LIN {X -0.214,Y -606.391,Z 470.276,A 0.000,B 0.000,C 90.000,E1 265.698} C_DIS
LIN {X -0.037,Y -603.397,Z 470.269,A 0.000,B 0.000,C 90.000,E1 264.375} C_DIS
LIN {X 0.001,Y -599.105,Z 470.259,A 0.000,B 0.000,C 90.000,E1 262.534} C_DIS
LIN {X 0.083,Y -594.642,Z 470.248,A 0.000,B 0.000,C 90.000,E1 260.679} C_DIS
LIN {X 0.202,Y -591.268,Z 470.241,A 0.000,B 0.000,C 90.000,E1 259.342} C_DIS
LIN {X -0.200,Y -587.770,Z 470.234,A 0.000,B 0.000,C 90.000,E1 258.049} C_DIS
LIN {X 0.160,Y -583.456,Z 470.225,A 0.000,B 0.000,C 90.000,E1 256.408} C_DIS
LIN {X -0.227,Y -579.823,Z 470.217,A 0.000,B 0.000,C 90.000,E1 255.102} C_DIS
LIN {X -0.114,Y -576.110,Z 470.210,A 0.000,B 0.000,C 90.000,E1 253.740} C_DIS
LIN {X -0.279,Y -571.459,Z 470.201,A 0.000,B 0.000,C 90.000,E1 252.127} C_DIS
LIN {X 0.013,Y -567.401,Z 470.193,A 0.000,B 0.000,C 90.000,E1 250.732} C_DIS
LIN {X -0.299,Y -563.218,Z 470.185,A 0.000,B 0.000,C 90.000,E1 249.390} C_DIS
LIN {X 0.041,Y -558.827,Z 470.178,A 0.000,B 0.000,C 90.000,E1 247.975} C_DIS
LIN {X 0.000,Y -555.124,Z 470.172,A 0.000,B 0.000,C 90.000,E1 246.869} C_DIS
LIN {X -0.109,Y -550.348,Z 470.164,A 0.000,B 0.000,C 90.000,E1 245.485} C_DIS
LIN {X 0.182,Y -544.388,Z 470.154,A 0.000,B 0.000,C 90.000,E1 243.768} C_DIS
LIN {X 0.121,Y -539.419,Z 470.147,A 0.000,B 0.000,C 90.000,E1 242.359} C_DIS
LIN {X -0.063,Y -533.493,Z 470.137,A 0.000,B 0.000,C 90.000,E1 240.667} C_DIS
LIN {X -0.149,Y -526.505,Z 470.126,A 0.000,B 0.000,C 90.000,E1 238.663} C_DIS
LIN {X -0.079,Y -520.654,Z 470.116,A 0.000,B 0.000,C 90.000,E1 236.914} C_DIS
LIN {X -0.224,Y -515.720,Z 470.108,A 0.000,B 0.000,C 90.000,E1 235.468} C_DIS
LIN {X -0.088,Y -511.559,Z 470.102,A 0.000,B 0.000,C 90.000,E1 234.276} C_DIS
LIN {X -0.248,Y -499.683,Z 470.082,A 0.000,B 0.000,C 90.000,E1 230.723} C_DIS
LIN {X 0.150,Y -493.420,Z 470.070,A 0.000,B 0.000,C 90.000,E1 228.566} C_DIS
LIN {X 0.119,Y -486.466,Z 470.056,A 0.000,B 0.000,C 90.000,E1 226.134} C_DIS
LIN {X 0.299,Y -481.414,Z 470.046,A 0.000,B 0.000,C 90.000,E1 224.271} C_DIS
LIN {X 0.135,Y -475.759,Z 470.034,A 0.000,B 0.000,C 90.000,E1 222.123} C_DIS
LIN {X -0.016,Y -469.737,Z 470.020,A 0.000,B 0.000,C 90.000,E1 219.644} C_DIS
LIN {X -0.034,Y -464.806,Z 470.008,A 0.000,B 0.000,C 90.000,E1 217.443} C_DIS
LIN {X 0.021,Y -459.483,Z 469.994,A 0.000,B 0.000,C 90.000,E1 214.898} C_DIS
LIN {X -0.076,Y -455.045,Z 469.982,A 0.000,B 0.000,C 90.000,E1 212.673} C_DIS
LIN {X 0.035,Y -452.006,Z 469.973,A 0.000,B 0.000,C 90.000,E1 211.052} C_DIS
LIN {X -0.209,Y -447.757,Z 469.960,A 0.000,B 0.000,C 90.000,E1 208.821} C_DIS
LIN {X -0.083,Y -444.730,Z 469.951,A 0.000,B 0.000,C 90.000,E1 207.180} C_DIS
LIN {X 0.123,Y -442.265,Z 469.944,A 0.000,B 0.000,C 90.000,E1 205.848} C_DIS
LIN {X -0.108,Y -439.798,Z 469.936,A 0.000,B 0.000,C 90.000,E1 204.567} C_DIS
LIN {X -0.086,Y -435.424,Z 469.924,A 0.000,B 0.000,C 90.000,E1 202.259} C_DIS
LIN {X -0.097,Y -431.263,Z 469.911,A 0.000,B 0.000,C 90.000,E1 199.939} C_DIS
LIN {X 0.051,Y -427.360,Z 469.898,A 0.000,B 0.000,C 90.000,E1 197.583} C_DIS
LIN {X 0.032,Y -423.295,Z 469.883,A 0.000,B 0.000,C 90.000,E1 194.898} C_DIS
LIN {X 0.017,Y -420.092,Z 469.870,A 0.000,B 0.000,C 90.000,E1 192.535} C_DIS
LIN {X -0.153,Y -416.381,Z 469.853,A 0.000,B 0.000,C 90.000,E1 189.500} C_DIS
LIN {X 0.142,Y -413.690,Z 469.839,A 0.000,B 0.000,C 90.000,E1 187.068} C_DIS
LIN {X -0.160,Y -412.241,Z 469.832,A 0.000,B 0.000,C 90.000,E1 185.739} C_DIS
LIN {X -0.118,Y -410.914,Z 469.824,A 0.000,B 0.000,C 90.000,E1 184.359} C_DIS
LIN {X -0.131,Y -408.830,Z 469.811,A 0.000,B 0.000,C 90.000,E1 181.949} C_DIS
LIN {X 0.156,Y -406.733,Z 469.793,A 0.000,B 0.000,C 90.000,E1 178.797} C_DIS
LIN {X -0.003,Y -405.511,Z 469.778,A 0.000,B 0.000,C 90.000,E1 176.045} C_DIS
LIN {X -0.104,Y -404.848,Z 469.763,A 0.000,B 0.000,C 90.000,E1 173.280} C_DIS
LIN {X -0.104,Y -404.977,Z 469.745,A 0.000,B 0.000,C 90.000,E1 170.151} C_DIS
LIN {X 0.123,Y -405.882,Z 469.728,A 0.000,B 0.000,C 90.000,E1 166.992} C_DIS
LIN {X 0.056,Y -407.044,Z 469.714,A 0.000,B 0.000,C 90.000,E1 164.574} C_DIS
LIN {X -0.061,Y -409.699,Z 469.693,A 0.000,B 0.000,C 90.000,E1 160.786} C_DIS
LIN {X 0.053,Y -411.869,Z 469.680,A 0.000,B 0.000,C 90.000,E1 158.358} C_DIS
LIN {X -0.079,Y -414.415,Z 469.667,A 0.000,B 0.000,C 90.000,E1 155.973} C_DIS
LIN {X -0.204,Y -416.381,Z 469.657,A 0.000,B 0.000,C 90.000,E1 154.280} C_DIS
LIN {X 0.107,Y -419.671,Z 469.642,A 0.000,B 0.000,C 90.000,E1 151.513} C_DIS
LIN {X 0.075,Y -421.752,Z 469.632,A 0.000,B 0.000,C 90.000,E1 149.822} C_DIS
LIN {X 0.146,Y -423.876,Z 469.623,A 0.000,B 0.000,C 90.000,E1 148.122} C_DIS
LIN {X -0.101,Y -426.458,Z 469.612,A 0.000,B 0.000,C 90.000,E1 146.135} C_DIS
LIN {X -0.048,Y -429.095,Z 469.601,A 0.000,B 0.000,C 90.000,E1 144.116} C_DIS
LIN {X 0.071,Y -430.982,Z 469.593,A 0.000,B 0.000,C 90.000,E1 142.763} C_DIS
LIN {X -0.214,Y -433.774,Z 469.582,A 0.000,B 0.000,C 90.000,E1 140.803} C_DIS
LIN {X -0.095,Y -435.681,Z 469.575,A 0.000,B 0.000,C 90.000,E1 139.461} C_DIS
LIN {X -0.003,Y -437.965,Z 469.566,A 0.000,B 0.000,C 90.000,E1 137.796} C_DIS
LIN {X 0.104,Y -440.095,Z 469.556,A 0.000,B 0.000,C 90.000,E1 136.134} C_DIS
LIN {X 0.001,Y -441.095,Z 469.551,A 0.000,B 0.000,C 90.000,E1 135.162} C_DIS
LIN {X -0.119,Y -442.209,Z 469.544,A 0.000,B 0.000,C 90.000,E1 133.866} C_DIS
LIN {X 0.095,Y -442.966,Z 469.536,A 0.000,B 0.000,C 90.000,E1 132.528} C_DIS
LIN {X 0.022,Y -443.267,Z 469.529,A 0.000,B 0.000,C 90.000,E1 131.229} C_DIS
LIN {X -0.017,Y -443.139,Z 469.524,A 0.000,B 0.000,C 90.000,E1 130.253} C_DIS
LIN {X -0.058,Y -442.518,Z 469.518,A 0.000,B 0.000,C 90.000,E1 129.277} C_DIS
LIN {X -0.110,Y -441.689,Z 469.513,A 0.000,B 0.000,C 90.000,E1 128.302} C_DIS
LIN {X -0.097,Y -440.525,Z 469.507,A 0.000,B 0.000,C 90.000,E1 127.317} C_DIS
LIN {X -0.155,Y -438.561,Z 469.500,A 0.000,B 0.000,C 90.000,E1 126.011} C_DIS
LIN {X 0.158,Y -437.427,Z 469.496,A 0.000,B 0.000,C 90.000,E1 125.311} C_DIS
LIN {X 0.148,Y -434.935,Z 469.489,A 0.000,B 0.000,C 90.000,E1 123.992} C_DIS
LIN {X 0.094,Y -432.035,Z 469.482,A 0.000,B 0.000,C 90.000,E1 122.673} C_DIS
LIN {X -0.005,Y -428.435,Z 469.473,A 0.000,B 0.000,C 90.000,E1 121.052} C_DIS
LIN {X -0.045,Y -428.429,Z 469.473,A 0.000,B 0.000,C 90.000,E1 121.052} C_DIS
LIN {X 0.121,Y -430.573,Z 469.469,A 0.000,B 0.000,C 90.000,E1 120.335} C_DIS
LIN {X -0.079,Y -441.483,Z 469.445,A 0.000,B 0.000,C 90.000,E1 116.052} C_DIS
LIN {X -0.159,Y -444.396,Z 469.439,A 0.000,B 0.000,C 90.000,E1 115.079} C_DIS
LIN {X 0.098,Y -445.208,Z 469.437,A 0.000,B 0.000,C 90.000,E1 114.719} C_DIS
LIN {X -0.040,Y -454.406,Z 469.416,A 0.000,B 0.000,C 90.000,E1 110.844} C_DIS
LIN {X -0.081,Y -457.079,Z 469.410,A 0.000,B 0.000,C 90.000,E1 109.885} C_DIS
LIN {X 0.004,Y -461.437,Z 469.398,A 0.000,B 0.000,C 90.000,E1 107.638} C_DIS
LIN {X -0.276,Y -467.270,Z 469.384,A 0.000,B 0.000,C 90.000,E1 105.134} C_DIS
LIN {X 0.101,Y -467.963,Z 469.382,A 0.000,B 0.000,C 90.000,E1 104.773} C_DIS
LIN {X -0.171,Y -476.219,Z 469.356,A 0.000,B 0.000,C 90.000,E1 100.074} C_DIS
LIN {X -0.091,Y -476.372,Z 469.355,A 0.000,B 0.000,C 90.000,E1 99.905} C_DIS
LIN {X -0.148,Y -526.605,Z 469.355,A 0.000,B 0.000,C 90.000,E1 99.905} C_DIS
LIN {X -0.102,Y -537.151,Z 469.355,A 0.000,B 0.000,C 90.000,E1 99.849} C_DIS
LIN {X 0.113,Y -540.500,Z 469.355,A 0.000,B 0.000,C 90.000,E1 99.792} C_DIS
LIN {X -0.208,Y -553.262,Z 469.353,A 0.000,B 0.000,C 90.000,E1 99.613} C_DIS
LIN {X 0.013,Y -559.633,Z 469.353,A 0.000,B 0.000,C 90.000,E1 99.443} C_DIS
LIN {X 0.063,Y -566.108,Z 469.352,A 0.000,B 0.000,C 90.000,E1 99.265} C_DIS
LIN {X 0.294,Y -576.120,Z 469.350,A 0.000,B 0.000,C 90.000,E1 98.916} C_DIS
LIN {X 0.150,Y -582.565,Z 469.348,A 0.000,B 0.000,C 90.000,E1 98.690} C_DIS
LIN {X 0.006,Y -592.233,Z 469.346,A 0.000,B 0.000,C 90.000,E1 98.276} C_DIS
LIN {X -0.304,Y -598.318,Z 469.344,A 0.000,B 0.000,C 90.000,E1 97.992} C_DIS
LIN {X -0.023,Y -601.041,Z 469.343,A 0.000,B 0.000,C 90.000,E1 97.814} C_DIS
LIN {X 0.102,Y -605.450,Z 469.342,A 0.000,B 0.000,C 90.000,E1 97.530} C_DIS
LIN {X 0.141,Y -611.163,Z 469.340,A 0.000,B 0.000,C 90.000,E1 97.125} C_DIS
LIN {X -0.132,Y -616.701,Z 469.337,A 0.000,B 0.000,C 90.000,E1 96.720} C_DIS
LIN {X -0.210,Y -623.076,Z 469.334,A 0.000,B 0.000,C 90.000,E1 96.144} C_DIS
LIN {X 0.323,Y -625.293,Z 469.333,A 0.000,B 0.000,C 90.000,E1 95.853} C_DIS
LIN {X -0.209,Y -629.691,Z 469.330,A 0.000,B 0.000,C 90.000,E1 95.391} C_DIS
LIN {X 0.002,Y -636.399,Z 469.324,A 0.000,B 0.000,C 90.000,E1 94.359} C_DIS
LIN {X 0.296,Y -638.500,Z 469.322,A 0.000,B 0.000,C 90.000,E1 93.955} C_DIS
LIN {X -0.083,Y -640.476,Z 469.320,A 0.000,B 0.000,C 90.000,E1 93.612} C_DIS
LIN {X 0.106,Y -642.677,Z 469.317,A 0.000,B 0.000,C 90.000,E1 93.094} C_DIS
LIN {X -0.135,Y -643.601,Z 469.316,A 0.000,B 0.000,C 90.000,E1 92.865} C_DIS
LIN {X 0.040,Y -645.162,Z 469.313,A 0.000,B 0.000,C 90.000,E1 92.350} C_DIS
LIN {X 0.232,Y -646.453,Z 469.310,A 0.000,B 0.000,C 90.000,E1 91.835} C_DIS
LIN {X -0.196,Y -647.322,Z 469.308,A 0.000,B 0.000,C 90.000,E1 91.375} C_DIS
LIN {X 0.010,Y -647.929,Z 469.305,A 0.000,B 0.000,C 90.000,E1 90.859} C_DIS
LIN {X -0.207,Y -648.173,Z 469.303,A 0.000,B 0.000,C 90.000,E1 90.630} C_DIS
LIN {X 0.008,Y -648.223,Z 469.301,A 0.000,B 0.000,C 90.000,E1 90.115} C_DIS
LIN {X 0.224,Y -647.934,Z 469.298,A 0.000,B 0.000,C 90.000,E1 89.599} C_DIS
LIN {X -0.209,Y -647.327,Z 469.295,A 0.000,B 0.000,C 90.000,E1 89.141} C_DIS
LIN {X 0.219,Y -646.938,Z 469.294,A 0.000,B 0.000,C 90.000,E1 88.854} C_DIS
LIN {X -0.221,Y -645.753,Z 469.291,A 0.000,B 0.000,C 90.000,E1 88.396} C_DIS
LIN {X -0.002,Y -644.242,Z 469.288,A 0.000,B 0.000,C 90.000,E1 87.879} C_DIS
LIN {X -0.228,Y -643.391,Z 469.287,A 0.000,B 0.000,C 90.000,E1 87.650} C_DIS
LIN {X -0.048,Y -641.396,Z 469.284,A 0.000,B 0.000,C 90.000,E1 87.135} C_DIS
LIN {X 0.151,Y -638.859,Z 469.281,A 0.000,B 0.000,C 90.000,E1 86.617} C_DIS
LIN {X 0.079,Y -634.722,Z 469.277,A 0.000,B 0.000,C 90.000,E1 85.869} C_DIS
LIN {X -0.173,Y -628.526,Z 469.272,A 0.000,B 0.000,C 90.000,E1 85.008} C_DIS
LIN {X -0.201,Y -623.501,Z 469.269,A 0.000,B 0.000,C 90.000,E1 84.375} C_DIS
LIN {X 0.184,Y -616.636,Z 469.264,A 0.000,B 0.000,C 90.000,E1 83.571} C_DIS
LIN {X -0.211,Y -611.344,Z 469.262,A 0.000,B 0.000,C 90.000,E1 83.109} C_DIS
LIN {X 0.221,Y -605.741,Z 469.259,A 0.000,B 0.000,C 90.000,E1 82.591} C_DIS
LIN {X -0.255,Y -599.923,Z 469.257,A 0.000,B 0.000,C 90.000,E1 82.186} C_DIS
LIN {X -0.109,Y -596.254,Z 469.255,A 0.000,B 0.000,C 90.000,E1 81.951} C_DIS
LIN {X -0.224,Y -593.898,Z 469.254,A 0.000,B 0.000,C 90.000,E1 81.781} C_DIS
LIN {X 0.017,Y -588.144,Z 469.252,A 0.000,B 0.000,C 90.000,E1 81.376} C_DIS
LIN {X -0.178,Y -584.150,Z 469.251,A 0.000,B 0.000,C 90.000,E1 81.197} C_DIS
LIN {X -0.046,Y -581.425,Z 469.250,A 0.000,B 0.000,C 90.000,E1 81.027} C_DIS
LIN {X -0.280,Y -575.599,Z 469.249,A 0.000,B 0.000,C 90.000,E1 80.792} C_DIS
LIN {X 0.043,Y -570.052,Z 469.248,A 0.000,B 0.000,C 90.000,E1 80.557} C_DIS
LIN {X 0.000,Y -563.805,Z 469.247,A 0.000,B 0.000,C 90.000,E1 80.387} C_DIS
LIN {X -0.304,Y -559.346,Z 469.246,A 0.000,B 0.000,C 90.000,E1 80.330} C_DIS
LIN {X -0.278,Y -556.297,Z 469.246,A 0.000,B 0.000,C 90.000,E1 80.274} C_DIS
LIN {X -0.067,Y -550.275,Z 469.246,A 0.000,B 0.000,C 90.000,E1 80.208} C_DIS
LIN {X -0.089,Y -483.137,Z 469.246,A 0.000,B 0.000,C 90.000,E1 80.208} C_DIS
LIN {X -0.081,Y -480.607,Z 469.228,A 0.000,B 0.000,C 90.000,E1 76.992} C_DIS
LIN {X -0.223,Y -480.245,Z 469.226,A 0.000,B 0.000,C 90.000,E1 76.700} C_DIS
LIN {X 0.134,Y -474.075,Z 469.200,A 0.000,B 0.000,C 90.000,E1 72.000} C_DIS
LIN {X 0.163,Y -465.515,Z 469.172,A 0.000,B 0.000,C 90.000,E1 66.975} C_DIS
LIN {X 0.094,Y -456.793,Z 469.148,A 0.000,B 0.000,C 90.000,E1 62.692} C_DIS
LIN {X 0.032,Y -456.650,Z 469.148,A 0.000,B 0.000,C 90.000,E1 62.615} C_DIS
LIN {X -0.008,Y -456.674,Z 469.148,A 0.000,B 0.000,C 90.000,E1 62.615} C_DIS
LIN {X 0.088,Y -465.116,Z 469.140,A 0.000,B 0.000,C 90.000,E1 61.257} C_DIS
LIN {X 0.137,Y -469.919,Z 469.136,A 0.000,B 0.000,C 90.000,E1 60.461} C_DIS
LIN {X 0.232,Y -474.530,Z 469.132,A 0.000,B 0.000,C 90.000,E1 59.665} C_DIS
LIN {X -0.035,Y -478.623,Z 469.127,A 0.000,B 0.000,C 90.000,E1 58.918} C_DIS
LIN {X -0.065,Y -480.940,Z 469.125,A 0.000,B 0.000,C 90.000,E1 58.456} C_DIS
LIN {X -0.050,Y -483.692,Z 469.121,A 0.000,B 0.000,C 90.000,E1 57.837} C_DIS
LIN {X -0.276,Y -486.044,Z 469.118,A 0.000,B 0.000,C 90.000,E1 57.248} C_DIS
LIN {X 0.007,Y -489.125,Z 469.113,A 0.000,B 0.000,C 90.000,E1 56.294} C_DIS
LIN {X -0.080,Y -491.318,Z 469.108,A 0.000,B 0.000,C 90.000,E1 55.388} C_DIS
LIN {X 0.010,Y -492.589,Z 469.104,A 0.000,B 0.000,C 90.000,E1 54.769} C_DIS
LIN {X -0.040,Y -494.001,Z 469.099,A 0.000,B 0.000,C 90.000,E1 53.863} C_DIS
LIN {X 0.216,Y -494.947,Z 469.094,A 0.000,B 0.000,C 90.000,E1 52.924} C_DIS
LIN {X 0.096,Y -495.629,Z 469.089,A 0.000,B 0.000,C 90.000,E1 52.029} C_DIS
LIN {X 0.066,Y -496.085,Z 469.084,A 0.000,B 0.000,C 90.000,E1 51.126} C_DIS
LIN {X -0.041,Y -496.341,Z 469.079,A 0.000,B 0.000,C 90.000,E1 50.231} C_DIS
LIN {X 0.179,Y -496.434,Z 469.074,A 0.000,B 0.000,C 90.000,E1 49.299} C_DIS
LIN {X 0.264,Y -496.318,Z 469.067,A 0.000,B 0.000,C 90.000,E1 48.081} C_DIS
LIN {X -0.209,Y -496.105,Z 469.062,A 0.000,B 0.000,C 90.000,E1 47.229} C_DIS
LIN {X 0.202,Y -495.692,Z 469.056,A 0.000,B 0.000,C 90.000,E1 45.972} C_DIS
LIN {X -0.263,Y -495.039,Z 469.047,A 0.000,B 0.000,C 90.000,E1 44.514} C_DIS
LIN {X -0.047,Y -494.218,Z 469.039,A 0.000,B 0.000,C 90.000,E1 42.975} C_DIS
LIN {X -0.157,Y -493.082,Z 469.030,A 0.000,B 0.000,C 90.000,E1 41.472} C_DIS
LIN {X 0.042,Y -491.981,Z 469.022,A 0.000,B 0.000,C 90.000,E1 39.930} C_DIS
LIN {X 0.118,Y -490.517,Z 469.012,A 0.000,B 0.000,C 90.000,E1 38.096} C_DIS
LIN {X 0.180,Y -489.507,Z 469.005,A 0.000,B 0.000,C 90.000,E1 36.870} C_DIS
LIN {X -0.064,Y -488.412,Z 468.998,A 0.000,B 0.000,C 90.000,E1 35.678} C_DIS
LIN {X -0.044,Y -487.237,Z 468.991,A 0.000,B 0.000,C 90.000,E1 34.452} C_DIS
LIN {X 0.042,Y -485.625,Z 468.983,A 0.000,B 0.000,C 90.000,E1 32.911} C_DIS
LIN {X 0.178,Y -483.531,Z 468.973,A 0.000,B 0.000,C 90.000,E1 31.052} C_DIS
LIN {X -0.261,Y -482.018,Z 468.966,A 0.000,B 0.000,C 90.000,E1 29.873} C_DIS
LIN {X 0.123,Y -479.814,Z 468.956,A 0.000,B 0.000,C 90.000,E1 27.975} C_DIS
LIN {X -0.223,Y -477.343,Z 468.944,A 0.000,B 0.000,C 90.000,E1 25.848} C_DIS
LIN {X -0.057,Y -474.460,Z 468.926,A 0.000,B 0.000,C 90.000,E1 22.717} C_DIS
LIN {X 0.121,Y -472.524,Z 468.911,A 0.000,B 0.000,C 90.000,E1 19.885} C_DIS
LIN {X 0.136,Y -471.211,Z 468.898,A 0.000,B 0.000,C 90.000,E1 17.692} C_DIS
LIN {X -0.128,Y -470.067,Z 468.888,A 0.000,B 0.000,C 90.000,E1 15.843} C_DIS
LIN {X 0.120,Y -468.728,Z 468.874,A 0.000,B 0.000,C 90.000,E1 13.300} C_DIS
LIN {X -0.251,Y -467.699,Z 468.857,A 0.000,B 0.000,C 90.000,E1 10.197} C_DIS
LIN {X 0.012,Y -467.337,Z 468.843,A 0.000,B 0.000,C 90.000,E1 7.644} C_DIS
LIN {X -0.078,Y -467.737,Z 468.823,A 0.000,B 0.000,C 90.000,E1 4.188} C_DIS
LIN {X 0.227,Y -469.374,Z 468.804,A 0.000,B 0.000,C 90.000,E1 0.688} C_DIS
LIN {X -0.218,Y -471.580,Z 468.788,A 0.000,B 0.000,C 90.000,E1 357.936} C_DIS
LIN {X -0.048,Y -474.192,Z 468.775,A 0.000,B 0.000,C 90.000,E1 355.412} C_DIS
LIN {X -0.151,Y -477.274,Z 468.761,A 0.000,B 0.000,C 90.000,E1 352.932} C_DIS
LIN {X 0.095,Y -481.700,Z 468.743,A 0.000,B 0.000,C 90.000,E1 349.803} C_DIS
LIN {X -0.184,Y -490.068,Z 468.718,A 0.000,B 0.000,C 90.000,E1 345.227} C_DIS
LIN {X -0.060,Y -495.409,Z 468.704,A 0.000,B 0.000,C 90.000,E1 342.779} C_DIS
LIN {X -0.063,Y -499.708,Z 468.694,A 0.000,B 0.000,C 90.000,E1 340.967} C_DIS
LIN {X 0.121,Y -503.389,Z 468.686,A 0.000,B 0.000,C 90.000,E1 339.444} C_DIS
LIN {X -0.103,Y -507.108,Z 468.678,A 0.000,B 0.000,C 90.000,E1 337.975} C_DIS
LIN {X -0.073,Y -510.736,Z 468.669,A 0.000,B 0.000,C 90.000,E1 336.485} C_DIS
LIN {X -0.213,Y -512.934,Z 468.664,A 0.000,B 0.000,C 90.000,E1 335.613} C_DIS
LIN {X 0.125,Y -516.463,Z 468.656,A 0.000,B 0.000,C 90.000,E1 334.101} C_DIS
LIN {X -0.166,Y -520.033,Z 468.648,A 0.000,B 0.000,C 90.000,E1 332.666} C_DIS
LIN {X 0.078,Y -523.580,Z 468.640,A 0.000,B 0.000,C 90.000,E1 331.179} C_DIS
LIN {X -0.126,Y -527.898,Z 468.630,A 0.000,B 0.000,C 90.000,E1 329.459} C_DIS
LIN {X 0.039,Y -532.324,Z 468.621,A 0.000,B 0.000,C 90.000,E1 327.709} C_DIS
LIN {X -0.153,Y -537.489,Z 468.610,A 0.000,B 0.000,C 90.000,E1 325.722} C_DIS
LIN {X 0.040,Y -541.224,Z 468.602,A 0.000,B 0.000,C 90.000,E1 324.276} C_DIS
LIN {X 0.208,Y -545.829,Z 468.592,A 0.000,B 0.000,C 90.000,E1 322.557} C_DIS
LIN {X 0.044,Y -550.377,Z 468.583,A 0.000,B 0.000,C 90.000,E1 320.884} C_DIS
LIN {X -0.101,Y -554.896,Z 468.573,A 0.000,B 0.000,C 90.000,E1 319.218} C_DIS
LIN {X 0.303,Y -560.197,Z 468.563,A 0.000,B 0.000,C 90.000,E1 317.229} C_DIS
LIN {X 0.013,Y -565.320,Z 468.552,A 0.000,B 0.000,C 90.000,E1 315.324} C_DIS
LIN {X -0.259,Y -569.637,Z 468.543,A 0.000,B 0.000,C 90.000,E1 313.704} C_DIS
LIN {X -0.248,Y -572.591,Z 468.537,A 0.000,B 0.000,C 90.000,E1 312.609} C_DIS
LIN {X 0.084,Y -576.826,Z 468.528,A 0.000,B 0.000,C 90.000,E1 310.943} C_DIS
LIN {X 0.064,Y -581.088,Z 468.519,A 0.000,B 0.000,C 90.000,E1 309.322} C_DIS
LIN {X -0.166,Y -585.312,Z 468.510,A 0.000,B 0.000,C 90.000,E1 307.729} C_DIS
LIN {X -0.033,Y -588.807,Z 468.502,A 0.000,B 0.000,C 90.000,E1 306.377} C_DIS
LIN {X 0.035,Y -592.869,Z 468.493,A 0.000,B 0.000,C 90.000,E1 304.771} C_DIS
LIN {X -0.036,Y -596.152,Z 468.486,A 0.000,B 0.000,C 90.000,E1 303.452} C_DIS
LIN {X -0.288,Y -598.661,Z 468.480,A 0.000,B 0.000,C 90.000,E1 302.418} C_DIS
LIN {X -0.004,Y -601.106,Z 468.474,A 0.000,B 0.000,C 90.000,E1 301.337} C_DIS
LIN {X 0.242,Y -603.935,Z 468.467,A 0.000,B 0.000,C 90.000,E1 300.001} C_DIS
LIN {X 0.293,Y -606.023,Z 468.461,A 0.000,B 0.000,C 90.000,E1 298.949} C_DIS
LIN {X 0.369,Y -607.930,Z 468.455,A 0.000,B 0.000,C 90.000,E1 297.897} C_DIS
LIN {X 0.066,Y -611.293,Z 468.445,A 0.000,B 0.000,C 90.000,E1 296.104} C_DIS
LIN {X -0.040,Y -612.586,Z 468.441,A 0.000,B 0.000,C 90.000,E1 295.335} C_DIS
LIN {X 0.107,Y -614.428,Z 468.434,A 0.000,B 0.000,C 90.000,E1 294.027} C_DIS
LIN {X 0.244,Y -616.844,Z 468.424,A 0.000,B 0.000,C 90.000,E1 292.206} C_DIS
LIN {X 0.236,Y -618.384,Z 468.416,A 0.000,B 0.000,C 90.000,E1 290.918} C_DIS
LIN {X 0.017,Y -620.101,Z 468.408,A 0.000,B 0.000,C 90.000,E1 289.396} C_DIS
LIN {X -0.174,Y -621.635,Z 468.399,A 0.000,B 0.000,C 90.000,E1 287.873} C_DIS
LIN {X 0.058,Y -623.055,Z 468.391,A 0.000,B 0.000,C 90.000,E1 286.315} C_DIS
LIN {X -0.245,Y -624.059,Z 468.384,A 0.000,B 0.000,C 90.000,E1 285.064} C_DIS
LIN {X 0.124,Y -624.729,Z 468.378,A 0.000,B 0.000,C 90.000,E1 284.008} C_DIS
LIN {X 0.101,Y -625.512,Z 468.369,A 0.000,B 0.000,C 90.000,E1 282.479} C_DIS
LIN {X 0.293,Y -625.911,Z 468.362,A 0.000,B 0.000,C 90.000,E1 281.186} C_DIS
LIN {X -0.252,Y -626.151,Z 468.355,A 0.000,B 0.000,C 90.000,E1 279.962} C_DIS
LIN {X 0.128,Y -625.966,Z 468.347,A 0.000,B 0.000,C 90.000,E1 278.398} C_DIS
LIN {X -0.215,Y -625.694,Z 468.341,A 0.000,B 0.000,C 90.000,E1 277.409} C_DIS
LIN {X 0.202,Y -625.319,Z 468.337,A 0.000,B 0.000,C 90.000,E1 276.606} C_DIS
LIN {X -0.231,Y -624.667,Z 468.331,A 0.000,B 0.000,C 90.000,E1 275.625} C_DIS
LIN {X 0.270,Y -623.439,Z 468.324,A 0.000,B 0.000,C 90.000,E1 274.302} C_DIS
LIN {X -0.241,Y -622.206,Z 468.318,A 0.000,B 0.000,C 90.000,E1 273.326} C_DIS
LIN {X -0.147,Y -620.769,Z 468.313,A 0.000,B 0.000,C 90.000,E1 272.293} C_DIS
LIN {X -0.079,Y -619.105,Z 468.307,A 0.000,B 0.000,C 90.000,E1 271.260} C_DIS
LIN {X 0.262,Y -616.863,Z 468.300,A 0.000,B 0.000,C 90.000,E1 269.943} C_DIS
LIN {X 0.246,Y -613.920,Z 468.291,A 0.000,B 0.000,C 90.000,E1 268.396} C_DIS
LIN {X 0.219,Y -611.803,Z 468.286,A 0.000,B 0.000,C 90.000,E1 267.364} C_DIS
LIN {X 0.166,Y -609.594,Z 468.280,A 0.000,B 0.000,C 90.000,E1 266.331} C_DIS
LIN {X -0.186,Y -607.893,Z 468.275,A 0.000,B 0.000,C 90.000,E1 265.584} C_DIS
LIN {X 0.014,Y -604.843,Z 468.268,A 0.000,B 0.000,C 90.000,E1 264.261} C_DIS
LIN {X -0.143,Y -601.122,Z 468.259,A 0.000,B 0.000,C 90.000,E1 262.704} C_DIS
LIN {X 0.294,Y -597.231,Z 468.251,A 0.000,B 0.000,C 90.000,E1 261.084} C_DIS
LIN {X -0.125,Y -593.897,Z 468.243,A 0.000,B 0.000,C 90.000,E1 259.803} C_DIS
LIN {X 0.249,Y -589.648,Z 468.234,A 0.000,B 0.000,C 90.000,E1 258.173} C_DIS
LIN {X 0.069,Y -585.249,Z 468.226,A 0.000,B 0.000,C 90.000,E1 256.589} C_DIS
LIN {X -0.063,Y -580.830,Z 468.217,A 0.000,B 0.000,C 90.000,E1 254.991} C_DIS
LIN {X -0.150,Y -577.822,Z 468.211,A 0.000,B 0.000,C 90.000,E1 253.921} C_DIS
LIN {X -0.280,Y -573.149,Z 468.202,A 0.000,B 0.000,C 90.000,E1 252.308} C_DIS
LIN {X -0.150,Y -568.232,Z 468.193,A 0.000,B 0.000,C 90.000,E1 250.659} C_DIS
LIN {X 0.090,Y -563.988,Z 468.185,A 0.000,B 0.000,C 90.000,E1 249.263} C_DIS
LIN {X -0.075,Y -559.589,Z 468.177,A 0.000,B 0.000,C 90.000,E1 247.901} C_DIS
LIN {X -0.098,Y -555.824,Z 468.171,A 0.000,B 0.000,C 90.000,E1 246.794} C_DIS
LIN {X -0.187,Y -551.005,Z 468.163,A 0.000,B 0.000,C 90.000,E1 245.409} C_DIS
LIN {X -0.115,Y -545.003,Z 468.154,A 0.000,B 0.000,C 90.000,E1 243.717} C_DIS
LIN {X 0.092,Y -541.007,Z 468.148,A 0.000,B 0.000,C 90.000,E1 242.564} C_DIS
LIN {X 0.197,Y -535.050,Z 468.138,A 0.000,B 0.000,C 90.000,E1 240.845} C_DIS
LIN {X 0.185,Y -529.009,Z 468.129,A 0.000,B 0.000,C 90.000,E1 239.125} C_DIS
LIN {X -0.063,Y -521.138,Z 468.116,A 0.000,B 0.000,C 90.000,E1 236.834} C_DIS
LIN {X -0.196,Y -516.196,Z 468.108,A 0.000,B 0.000,C 90.000,E1 235.388} C_DIS
LIN {X -0.127,Y -510.971,Z 468.099,A 0.000,B 0.000,C 90.000,E1 233.909} C_DIS
LIN {X -0.306,Y -499.239,Z 468.080,A 0.000,B 0.000,C 90.000,E1 230.356} C_DIS
LIN {X -0.143,Y -493.865,Z 468.070,A 0.000,B 0.000,C 90.000,E1 228.528} C_DIS
LIN {X 0.210,Y -486.936,Z 468.056,A 0.000,B 0.000,C 90.000,E1 226.053} C_DIS
LIN {X -0.282,Y -481.901,Z 468.046,A 0.000,B 0.000,C 90.000,E1 224.271} C_DIS
LIN {X 0.035,Y -475.440,Z 468.032,A 0.000,B 0.000,C 90.000,E1 221.757} C_DIS
LIN {X 0.105,Y -470.205,Z 468.020,A 0.000,B 0.000,C 90.000,E1 219.564} C_DIS
LIN {X 0.097,Y -465.261,Z 468.008,A 0.000,B 0.000,C 90.000,E1 217.363} C_DIS
LIN {X 0.039,Y -460.593,Z 467.995,A 0.000,B 0.000,C 90.000,E1 215.152} C_DIS
LIN {X -0.287,Y -456.091,Z 467.983,A 0.000,B 0.000,C 90.000,E1 212.959} C_DIS
LIN {X -0.051,Y -452.410,Z 467.972,A 0.000,B 0.000,C 90.000,E1 211.003} C_DIS
LIN {X -0.136,Y -448.780,Z 467.961,A 0.000,B 0.000,C 90.000,E1 209.077} C_DIS
LIN {X -0.134,Y -445.153,Z 467.951,A 0.000,B 0.000,C 90.000,E1 207.129} C_DIS
LIN {X 0.128,Y -442.052,Z 467.942,A 0.000,B 0.000,C 90.000,E1 205.463} C_DIS
LIN {X 0.134,Y -438.893,Z 467.932,A 0.000,B 0.000,C 90.000,E1 203.823} C_DIS
LIN {X -0.029,Y -434.559,Z 467.920,A 0.000,B 0.000,C 90.000,E1 201.535} C_DIS
LIN {X 0.130,Y -430.992,Z 467.909,A 0.000,B 0.000,C 90.000,E1 199.523} C_DIS
LIN {X 0.198,Y -427.662,Z 467.897,A 0.000,B 0.000,C 90.000,E1 197.511} C_DIS
LIN {X 0.174,Y -423.572,Z 467.883,A 0.000,B 0.000,C 90.000,E1 194.828} C_DIS
LIN {X -0.009,Y -420.793,Z 467.871,A 0.000,B 0.000,C 90.000,E1 192.827} C_DIS
LIN {X -0.155,Y -417.027,Z 467.854,A 0.000,B 0.000,C 90.000,E1 189.792} C_DIS
LIN {X 0.216,Y -414.290,Z 467.841,A 0.000,B 0.000,C 90.000,E1 187.352} C_DIS
LIN {X -0.089,Y -412.479,Z 467.832,A 0.000,B 0.000,C 90.000,E1 185.682} C_DIS
LIN {X -0.029,Y -410.479,Z 467.820,A 0.000,B 0.000,C 90.000,E1 183.612} C_DIS
LIN {X -0.060,Y -408.513,Z 467.807,A 0.000,B 0.000,C 90.000,E1 181.203} C_DIS
LIN {X 0.196,Y -406.406,Z 467.787,A 0.000,B 0.000,C 90.000,E1 177.707} C_DIS
LIN {X 0.058,Y -405.485,Z 467.774,A 0.000,B 0.000,C 90.000,E1 175.298} C_DIS
LIN {X -0.029,Y -405.073,Z 467.753,A 0.000,B 0.000,C 90.000,E1 171.489} C_DIS
LIN {X 0.117,Y -405.657,Z 467.735,A 0.000,B 0.000,C 90.000,E1 168.342} C_DIS
LIN {X 0.060,Y -407.016,Z 467.718,A 0.000,B 0.000,C 90.000,E1 165.227} C_DIS
LIN {X -0.186,Y -409.477,Z 467.697,A 0.000,B 0.000,C 90.000,E1 161.456} C_DIS
LIN {X -0.076,Y -411.606,Z 467.683,A 0.000,B 0.000,C 90.000,E1 159.028} C_DIS
LIN {X -0.130,Y -413.707,Z 467.672,A 0.000,B 0.000,C 90.000,E1 156.975} C_DIS
LIN {X 0.178,Y -416.475,Z 467.659,A 0.000,B 0.000,C 90.000,E1 154.537} C_DIS
LIN {X -0.074,Y -419.770,Z 467.644,A 0.000,B 0.000,C 90.000,E1 151.847} C_DIS
LIN {X 0.104,Y -421.897,Z 467.634,A 0.000,B 0.000,C 90.000,E1 150.127} C_DIS
LIN {X -0.079,Y -424.935,Z 467.621,A 0.000,B 0.000,C 90.000,E1 147.788} C_DIS
LIN {X 0.049,Y -427.605,Z 467.610,A 0.000,B 0.000,C 90.000,E1 145.754} C_DIS
LIN {X 0.014,Y -430.884,Z 467.597,A 0.000,B 0.000,C 90.000,E1 143.417} C_DIS
LIN {X -0.010,Y -434.217,Z 467.584,A 0.000,B 0.000,C 90.000,E1 141.090} C_DIS
LIN {X -0.223,Y -436.669,Z 467.575,A 0.000,B 0.000,C 90.000,E1 139.461} C_DIS
LIN {X -0.111,Y -439.101,Z 467.565,A 0.000,B 0.000,C 90.000,E1 137.796} C_DIS
LIN {X 0.018,Y -441.323,Z 467.556,A 0.000,B 0.000,C 90.000,E1 136.134} C_DIS
LIN {X -0.097,Y -442.713,Z 467.549,A 0.000,B 0.000,C 90.000,E1 134.838} C_DIS
LIN {X -0.147,Y -443.338,Z 467.545,A 0.000,B 0.000,C 90.000,E1 134.190} C_DIS
LIN {X 0.108,Y -444.040,Z 467.540,A 0.000,B 0.000,C 90.000,E1 133.176} C_DIS
LIN {X 0.045,Y -444.514,Z 467.535,A 0.000,B 0.000,C 90.000,E1 132.204} C_DIS
LIN {X 0.015,Y -444.787,Z 467.529,A 0.000,B 0.000,C 90.000,E1 131.229} C_DIS
LIN {X -0.007,Y -444.703,Z 467.524,A 0.000,B 0.000,C 90.000,E1 130.253} C_DIS
LIN {X -0.060,Y -443.919,Z 467.516,A 0.000,B 0.000,C 90.000,E1 128.955} C_DIS
LIN {X -0.025,Y -443.006,Z 467.511,A 0.000,B 0.000,C 90.000,E1 127.971} C_DIS
LIN {X -0.077,Y -441.762,Z 467.506,A 0.000,B 0.000,C 90.000,E1 126.996} C_DIS
LIN {X -0.060,Y -440.315,Z 467.500,A 0.000,B 0.000,C 90.000,E1 126.011} C_DIS
LIN {X -0.090,Y -439.161,Z 467.496,A 0.000,B 0.000,C 90.000,E1 125.358} C_DIS
LIN {X -0.079,Y -436.596,Z 467.489,A 0.000,B 0.000,C 90.000,E1 124.040} C_DIS
LIN {X -0.002,Y -434.413,Z 467.484,A 0.000,B 0.000,C 90.000,E1 123.038} C_DIS
LIN {X -0.057,Y -430.655,Z 467.474,A 0.000,B 0.000,C 90.000,E1 121.386} C_DIS
LIN {X -0.127,Y -429.254,Z 467.471,A 0.000,B 0.000,C 90.000,E1 120.797} C_DIS
LIN {X -0.166,Y -429.257,Z 467.471,A 0.000,B 0.000,C 90.000,E1 120.797} C_DIS
LIN {X -0.048,Y -430.488,Z 467.469,A 0.000,B 0.000,C 90.000,E1 120.384} C_DIS
LIN {X -0.255,Y -432.832,Z 467.463,A 0.000,B 0.000,C 90.000,E1 119.411} C_DIS
LIN {X 0.160,Y -442.358,Z 467.443,A 0.000,B 0.000,C 90.000,E1 115.720} C_DIS
LIN {X 0.045,Y -444.316,Z 467.439,A 0.000,B 0.000,C 90.000,E1 115.079} C_DIS
LIN {X -0.101,Y -445.154,Z 467.438,A 0.000,B 0.000,C 90.000,E1 114.771} C_DIS
LIN {X 0.005,Y -454.336,Z 467.416,A 0.000,B 0.000,C 90.000,E1 110.865} C_DIS
LIN {X 0.126,Y -457.005,Z 467.411,A 0.000,B 0.000,C 90.000,E1 109.885} C_DIS
LIN {X -0.066,Y -458.258,Z 467.407,A 0.000,B 0.000,C 90.000,E1 109.268} C_DIS
LIN {X 0.132,Y -466.422,Z 467.386,A 0.000,B 0.000,C 90.000,E1 105.426} C_DIS
LIN {X -0.145,Y -467.928,Z 467.382,A 0.000,B 0.000,C 90.000,E1 104.828} C_DIS
LIN {X -0.031,Y -475.504,Z 467.358,A 0.000,B 0.000,C 90.000,E1 100.423} C_DIS
LIN {X 0.189,Y -476.143,Z 467.356,A 0.000,B 0.000,C 90.000,E1 100.084} C_DIS
LIN {X -0.008,Y -476.878,Z 467.352,A 0.000,B 0.000,C 90.000,E1 99.378} C_DIS
LIN {X -0.056,Y -530.973,Z 467.352,A 0.000,B 0.000,C 90.000,E1 99.378} C_DIS
LIN {X -0.190,Y -537.802,Z 467.352,A 0.000,B 0.000,C 90.000,E1 99.378} C_DIS
LIN {X -0.096,Y -543.434,Z 467.352,A 0.000,B 0.000,C 90.000,E1 99.321} C_DIS
LIN {X 0.076,Y -550.690,Z 467.351,A 0.000,B 0.000,C 90.000,E1 99.208} C_DIS
LIN {X 0.194,Y -556.636,Z 467.351,A 0.000,B 0.000,C 90.000,E1 99.095} C_DIS
LIN {X -0.017,Y -562.880,Z 467.350,A 0.000,B 0.000,C 90.000,E1 98.973} C_DIS
LIN {X -0.131,Y -569.279,Z 467.349,A 0.000,B 0.000,C 90.000,E1 98.803} C_DIS
LIN {X 0.126,Y -579.416,Z 467.347,A 0.000,B 0.000,C 90.000,E1 98.454} C_DIS
LIN {X 0.088,Y -590.622,Z 467.345,A 0.000,B 0.000,C 90.000,E1 97.992} C_DIS
LIN {X -0.059,Y -592.327,Z 467.344,A 0.000,B 0.000,C 90.000,E1 97.936} C_DIS
LIN {X -0.174,Y -598.461,Z 467.342,A 0.000,B 0.000,C 90.000,E1 97.644} C_DIS
LIN {X -0.100,Y -604.433,Z 467.341,A 0.000,B 0.000,C 90.000,E1 97.296} C_DIS
LIN {X 0.122,Y -610.058,Z 467.338,A 0.000,B 0.000,C 90.000,E1 96.891} C_DIS
LIN {X -0.068,Y -616.983,Z 467.335,A 0.000,B 0.000,C 90.000,E1 96.372} C_DIS
LIN {X -0.213,Y -623.365,Z 467.332,A 0.000,B 0.000,C 90.000,E1 95.796} C_DIS
LIN {X 0.124,Y -626.588,Z 467.330,A 0.000,B 0.000,C 90.000,E1 95.391} C_DIS
LIN {X -0.025,Y -627.569,Z 467.329,A 0.000,B 0.000,C 90.000,E1 95.277} C_DIS
LIN {X -0.105,Y -628.775,Z 467.329,A 0.000,B 0.000,C 90.000,E1 95.163} C_DIS
LIN {X -0.185,Y -629.743,Z 467.328,A 0.000,B 0.000,C 90.000,E1 95.049} C_DIS
LIN {X 0.167,Y -635.679,Z 467.323,A 0.000,B 0.000,C 90.000,E1 94.131} C_DIS
LIN {X 0.201,Y -638.802,Z 467.320,A 0.000,B 0.000,C 90.000,E1 93.498} C_DIS
LIN {X -0.172,Y -640.501,Z 467.317,A 0.000,B 0.000,C 90.000,E1 93.154} C_DIS
LIN {X -0.261,Y -641.123,Z 467.317,A 0.000,B 0.000,C 90.000,E1 93.037} C_DIS
LIN {X -0.104,Y -642.797,Z 467.314,A 0.000,B 0.000,C 90.000,E1 92.522} C_DIS
LIN {X -0.141,Y -644.738,Z 467.310,A 0.000,B 0.000,C 90.000,E1 91.776} C_DIS
LIN {X 0.046,Y -645.539,Z 467.307,A 0.000,B 0.000,C 90.000,E1 91.260} C_DIS
LIN {X 0.241,Y -646.088,Z 467.304,A 0.000,B 0.000,C 90.000,E1 90.745} C_DIS
LIN {X -0.205,Y -646.238,Z 467.302,A 0.000,B 0.000,C 90.000,E1 90.286} C_DIS
LIN {X 0.219,Y -646.234,Z 467.300,A 0.000,B 0.000,C 90.000,E1 90.000} C_DIS
LIN {X -0.224,Y -645.863,Z 467.297,A 0.000,B 0.000,C 90.000,E1 89.542} C_DIS
LIN {X -0.025,Y -645.108,Z 467.295,A 0.000,B 0.000,C 90.000,E1 89.026} C_DIS
LIN {X 0.169,Y -644.033,Z 467.292,A 0.000,B 0.000,C 90.000,E1 88.511} C_DIS
LIN {X -0.059,Y -643.427,Z 467.290,A 0.000,B 0.000,C 90.000,E1 88.282} C_DIS
LIN {X 0.145,Y -641.908,Z 467.288,A 0.000,B 0.000,C 90.000,E1 87.764} C_DIS
LIN {X -0.090,Y -640.958,Z 467.286,A 0.000,B 0.000,C 90.000,E1 87.535} C_DIS
LIN {X -0.139,Y -637.141,Z 467.282,A 0.000,B 0.000,C 90.000,E1 86.788} C_DIS
LIN {X -0.009,Y -634.433,Z 467.279,A 0.000,B 0.000,C 90.000,E1 86.274} C_DIS
LIN {X -0.265,Y -628.548,Z 467.274,A 0.000,B 0.000,C 90.000,E1 85.412} C_DIS
LIN {X 0.177,Y -622.556,Z 467.270,A 0.000,B 0.000,C 90.000,E1 84.609} C_DIS
LIN {X 0.156,Y -616.780,Z 467.267,A 0.000,B 0.000,C 90.000,E1 83.970} C_DIS
LIN {X 0.250,Y -611.620,Z 467.264,A 0.000,B 0.000,C 90.000,E1 83.457} C_DIS
LIN {X -0.048,Y -605.065,Z 467.261,A 0.000,B 0.000,C 90.000,E1 82.932} C_DIS
LIN {X 0.211,Y -599.017,Z 467.258,A 0.000,B 0.000,C 90.000,E1 82.470} C_DIS
LIN {X -0.220,Y -586.564,Z 467.254,A 0.000,B 0.000,C 90.000,E1 81.724} C_DIS
LIN {X 0.052,Y -581.346,Z 467.252,A 0.000,B 0.000,C 90.000,E1 81.432} C_DIS
LIN {X 0.027,Y -575.821,Z 467.251,A 0.000,B 0.000,C 90.000,E1 81.197} C_DIS
LIN {X -0.124,Y -574.011,Z 467.251,A 0.000,B 0.000,C 90.000,E1 81.141} C_DIS
LIN {X -0.315,Y -567.758,Z 467.250,A 0.000,B 0.000,C 90.000,E1 80.971} C_DIS
LIN {X 0.093,Y -561.436,Z 467.249,A 0.000,B 0.000,C 90.000,E1 80.792} C_DIS
LIN {X -0.180,Y -555.067,Z 467.248,A 0.000,B 0.000,C 90.000,E1 80.735} C_DIS
LIN {X 0.106,Y -549.476,Z 467.248,A 0.000,B 0.000,C 90.000,E1 80.679} C_DIS
LIN {X 0.056,Y -483.660,Z 467.248,A 0.000,B 0.000,C 90.000,E1 80.679} C_DIS
LIN {X -0.135,Y -480.603,Z 467.228,A 0.000,B 0.000,C 90.000,E1 76.992} C_DIS
LIN {X 0.190,Y -480.234,Z 467.226,A 0.000,B 0.000,C 90.000,E1 76.645} C_DIS
LIN {X 0.081,Y -474.065,Z 467.200,A 0.000,B 0.000,C 90.000,E1 72.000} C_DIS
LIN {X 0.109,Y -465.499,Z 467.172,A 0.000,B 0.000,C 90.000,E1 66.975} C_DIS
LIN {X -0.151,Y -457.046,Z 467.149,A 0.000,B 0.000,C 90.000,E1 62.871} C_DIS
LIN {X -0.192,Y -457.048,Z 467.149,A 0.000,B 0.000,C 90.000,E1 62.871} C_DIS
LIN {X 0.267,Y -462.048,Z 467.145,A 0.000,B 0.000,C 90.000,E1 62.025} C_DIS
LIN {X -0.163,Y -468.106,Z 467.140,A 0.000,B 0.000,C 90.000,E1 61.129} C_DIS
LIN {X -0.152,Y -475.641,Z 467.133,A 0.000,B 0.000,C 90.000,E1 59.871} C_DIS
LIN {X -0.005,Y -479.805,Z 467.128,A 0.000,B 0.000,C 90.000,E1 59.076} C_DIS
LIN {X -0.027,Y -482.142,Z 467.126,A 0.000,B 0.000,C 90.000,E1 58.614} C_DIS
LIN {X -0.231,Y -485.538,Z 467.121,A 0.000,B 0.000,C 90.000,E1 57.867} C_DIS
LIN {X -0.186,Y -487.898,Z 467.118,A 0.000,B 0.000,C 90.000,E1 57.248} C_DIS
LIN {X -0.120,Y -489.930,Z 467.115,A 0.000,B 0.000,C 90.000,E1 56.628} C_DIS
LIN {X -0.039,Y -491.634,Z 467.111,A 0.000,B 0.000,C 90.000,E1 56.008} C_DIS
LIN {X 0.211,Y -492.395,Z 467.109,A 0.000,B 0.000,C 90.000,E1 55.674} C_DIS
LIN {X 0.159,Y -494.223,Z 467.104,A 0.000,B 0.000,C 90.000,E1 54.769} C_DIS
LIN {X -0.131,Y -495.181,Z 467.101,A 0.000,B 0.000,C 90.000,E1 54.196} C_DIS
LIN {X 0.143,Y -496.267,Z 467.096,A 0.000,B 0.000,C 90.000,E1 53.256} C_DIS
LIN {X 0.131,Y -496.984,Z 467.091,A 0.000,B 0.000,C 90.000,E1 52.351} C_DIS
LIN {X 0.034,Y -497.459,Z 467.086,A 0.000,B 0.000,C 90.000,E1 51.457} C_DIS
LIN {X -0.185,Y -497.742,Z 467.079,A 0.000,B 0.000,C 90.000,E1 50.275} C_DIS
LIN {X -0.134,Y -497.819,Z 467.076,A 0.000,B 0.000,C 90.000,E1 49.666} C_DIS
LIN {X -0.025,Y -497.647,Z 467.069,A 0.000,B 0.000,C 90.000,E1 48.447} C_DIS
LIN {X -0.115,Y -497.432,Z 467.064,A 0.000,B 0.000,C 90.000,E1 47.553} C_DIS
LIN {X -0.194,Y -496.861,Z 467.056,A 0.000,B 0.000,C 90.000,E1 46.053} C_DIS
LIN {X 0.063,Y -496.124,Z 467.047,A 0.000,B 0.000,C 90.000,E1 44.514} C_DIS
LIN {X -0.039,Y -495.259,Z 467.039,A 0.000,B 0.000,C 90.000,E1 43.014} C_DIS
LIN {X -0.163,Y -494.089,Z 467.031,A 0.000,B 0.000,C 90.000,E1 41.515} C_DIS
LIN {X -0.269,Y -492.975,Z 467.022,A 0.000,B 0.000,C 90.000,E1 40.011} C_DIS
LIN {X -0.016,Y -491.707,Z 467.014,A 0.000,B 0.000,C 90.000,E1 38.463} C_DIS
LIN {X 0.063,Y -490.726,Z 467.007,A 0.000,B 0.000,C 90.000,E1 37.237} C_DIS
LIN {X -0.031,Y -489.365,Z 466.999,A 0.000,B 0.000,C 90.000,E1 35.724} C_DIS
LIN {X 0.124,Y -488.150,Z 466.992,A 0.000,B 0.000,C 90.000,E1 34.485} C_DIS
LIN {X -0.141,Y -486.871,Z 466.985,A 0.000,B 0.000,C 90.000,E1 33.293} C_DIS
LIN {X -0.054,Y -485.096,Z 466.976,A 0.000,B 0.000,C 90.000,E1 31.750} C_DIS
LIN {X -0.219,Y -483.687,Z 466.970,A 0.000,B 0.000,C 90.000,E1 30.541} C_DIS
LIN {X -0.002,Y -481.023,Z 466.958,A 0.000,B 0.000,C 90.000,E1 28.359} C_DIS
LIN {X 0.129,Y -478.826,Z 466.947,A 0.000,B 0.000,C 90.000,E1 26.488} C_DIS
LIN {X 0.104,Y -475.755,Z 466.930,A 0.000,B 0.000,C 90.000,E1 23.387} C_DIS
LIN {X -0.097,Y -473.859,Z 466.916,A 0.000,B 0.000,C 90.000,E1 20.918} C_DIS
LIN {X -0.006,Y -472.652,Z 466.906,A 0.000,B 0.000,C 90.000,E1 19.033} C_DIS
LIN {X 0.096,Y -471.784,Z 466.897,A 0.000,B 0.000,C 90.000,E1 17.457} C_DIS
LIN {X 0.244,Y -470.414,Z 466.885,A 0.000,B 0.000,C 90.000,E1 15.245} C_DIS
LIN {X 0.113,Y -469.226,Z 466.873,A 0.000,B 0.000,C 90.000,E1 13.063} C_DIS
LIN {X 0.127,Y -468.370,Z 466.859,A 0.000,B 0.000,C 90.000,E1 10.546} C_DIS
LIN {X -0.052,Y -467.937,Z 466.845,A 0.000,B 0.000,C 90.000,E1 8.049} C_DIS
LIN {X 0.151,Y -468.241,Z 466.824,A 0.000,B 0.000,C 90.000,E1 4.245} C_DIS
LIN {X 0.006,Y -469.792,Z 466.805,A 0.000,B 0.000,C 90.000,E1 0.802} C_DIS
LIN {X -0.207,Y -472.049,Z 466.788,A 0.000,B 0.000,C 90.000,E1 357.936} C_DIS
LIN {X 0.197,Y -474.307,Z 466.776,A 0.000,B 0.000,C 90.000,E1 355.698} C_DIS
LIN {X 0.051,Y -477.285,Z 466.762,A 0.000,B 0.000,C 90.000,E1 353.223} C_DIS
LIN {X -0.221,Y -480.260,Z 466.750,A 0.000,B 0.000,C 90.000,E1 351.084} C_DIS
LIN {X 0.014,Y -482.649,Z 466.742,A 0.000,B 0.000,C 90.000,E1 349.511} C_DIS
LIN {X -0.098,Y -490.561,Z 466.718,A 0.000,B 0.000,C 90.000,E1 345.227} C_DIS
LIN {X 0.040,Y -495.899,Z 466.704,A 0.000,B 0.000,C 90.000,E1 342.779} C_DIS
LIN {X 0.050,Y -500.194,Z 466.694,A 0.000,B 0.000,C 90.000,E1 340.967} C_DIS
LIN {X 0.165,Y -503.214,Z 466.688,A 0.000,B 0.000,C 90.000,E1 339.752} C_DIS
LIN {X 0.032,Y -507.681,Z 466.678,A 0.000,B 0.000,C 90.000,E1 337.975} C_DIS
LIN {X 0.182,Y -512.093,Z 466.668,A 0.000,B 0.000,C 90.000,E1 336.177} C_DIS
LIN {X 0.044,Y -515.739,Z 466.660,A 0.000,B 0.000,C 90.000,E1 334.717} C_DIS
LIN {X 0.013,Y -520.726,Z 466.648,A 0.000,B 0.000,C 90.000,E1 332.666} C_DIS
LIN {X -0.046,Y -525.037,Z 466.638,A 0.000,B 0.000,C 90.000,E1 330.923} C_DIS
LIN {X 0.087,Y -528.693,Z 466.630,A 0.000,B 0.000,C 90.000,E1 329.459} C_DIS
LIN {X 0.289,Y -532.407,Z 466.622,A 0.000,B 0.000,C 90.000,E1 327.995} C_DIS
LIN {X 0.099,Y -536.089,Z 466.614,A 0.000,B 0.000,C 90.000,E1 326.580} C_DIS
LIN {X -0.181,Y -539.867,Z 466.607,A 0.000,B 0.000,C 90.000,E1 325.182} C_DIS
LIN {X -0.008,Y -545.190,Z 466.595,A 0.000,B 0.000,C 90.000,E1 323.176} C_DIS
LIN {X 0.255,Y -549.814,Z 466.586,A 0.000,B 0.000,C 90.000,E1 321.457} C_DIS
LIN {X -0.252,Y -554.380,Z 466.577,A 0.000,B 0.000,C 90.000,E1 319.828} C_DIS
LIN {X 0.138,Y -559.692,Z 466.566,A 0.000,B 0.000,C 90.000,E1 317.838} C_DIS
LIN {X -0.040,Y -561.962,Z 466.561,A 0.000,B 0.000,C 90.000,E1 317.025} C_DIS
LIN {X 0.016,Y -566.465,Z 466.552,A 0.000,B 0.000,C 90.000,E1 315.364} C_DIS
LIN {X -0.333,Y -570.111,Z 466.544,A 0.000,B 0.000,C 90.000,E1 314.028} C_DIS
LIN {X 0.075,Y -573.104,Z 466.538,A 0.000,B 0.000,C 90.000,E1 312.894} C_DIS
LIN {X -0.114,Y -576.734,Z 466.531,A 0.000,B 0.000,C 90.000,E1 311.553} C_DIS
LIN {X -0.130,Y -581.028,Z 466.522,A 0.000,B 0.000,C 90.000,E1 309.930} C_DIS
LIN {X 0.282,Y -584.645,Z 466.514,A 0.000,B 0.000,C 90.000,E1 308.543} C_DIS
LIN {X 0.137,Y -588.859,Z 466.505,A 0.000,B 0.000,C 90.000,E1 306.950} C_DIS
LIN {X -0.144,Y -592.331,Z 466.498,A 0.000,B 0.000,C 90.000,E1 305.644} C_DIS
LIN {X 0.034,Y -595.030,Z 466.492,A 0.000,B 0.000,C 90.000,E1 304.565} C_DIS
LIN {X -0.124,Y -597.056,Z 466.488,A 0.000,B 0.000,C 90.000,E1 303.785} C_DIS
LIN {X -0.136,Y -600.187,Z 466.480,A 0.000,B 0.000,C 90.000,E1 302.467} C_DIS
LIN {X 0.090,Y -603.186,Z 466.473,A 0.000,B 0.000,C 90.000,E1 301.131} C_DIS
LIN {X 0.129,Y -605.483,Z 466.467,A 0.000,B 0.000,C 90.000,E1 300.079} C_DIS
LIN {X -0.328,Y -607.570,Z 466.461,A 0.000,B 0.000,C 90.000,E1 299.077} C_DIS
LIN {X -0.186,Y -609.054,Z 466.457,A 0.000,B 0.000,C 90.000,E1 298.281} C_DIS
LIN {X 0.048,Y -612.945,Z 466.446,A 0.000,B 0.000,C 90.000,E1 296.181} C_DIS
LIN {X 0.018,Y -613.289,Z 466.444,A 0.000,B 0.000,C 90.000,E1 295.924} C_DIS
LIN {X -0.039,Y -614.271,Z 466.441,A 0.000,B 0.000,C 90.000,E1 295.412} C_DIS
LIN {X -0.166,Y -616.189,Z 466.434,A 0.000,B 0.000,C 90.000,E1 294.131} C_DIS
LIN {X -0.236,Y -618.698,Z 466.424,A 0.000,B 0.000,C 90.000,E1 292.333} C_DIS
LIN {X -0.213,Y -620.296,Z 466.417,A 0.000,B 0.000,C 90.000,E1 291.046} C_DIS
LIN {X -0.183,Y -622.052,Z 466.408,A 0.000,B 0.000,C 90.000,E1 289.504} C_DIS
LIN {X 0.055,Y -623.622,Z 466.400,A 0.000,B 0.000,C 90.000,E1 287.946} C_DIS
LIN {X -0.049,Y -624.870,Z 466.393,A 0.000,B 0.000,C 90.000,E1 286.677} C_DIS
LIN {X 0.081,Y -626.128,Z 466.384,A 0.000,B 0.000,C 90.000,E1 285.134} C_DIS
LIN {X -0.171,Y -626.975,Z 466.377,A 0.000,B 0.000,C 90.000,E1 283.883} C_DIS
LIN {X 0.043,Y -627.609,Z 466.370,A 0.000,B 0.000,C 90.000,E1 282.591} C_DIS
LIN {X 0.266,Y -628.068,Z 466.363,A 0.000,B 0.000,C 90.000,E1 281.299} C_DIS
LIN {X -0.045,Y -628.290,Z 466.357,A 0.000,B 0.000,C 90.000,E1 280.310} C_DIS
LIN {X 0.269,Y -628.257,Z 466.352,A 0.000,B 0.000,C 90.000,E1 279.265} C_DIS
LIN {X -0.041,Y -628.139,Z 466.346,A 0.000,B 0.000,C 90.000,E1 278.276} C_DIS
LIN {X -0.229,Y -627.921,Z 466.342,A 0.000,B 0.000,C 90.000,E1 277.530} C_DIS
LIN {X 0.070,Y -627.401,Z 466.336,A 0.000,B 0.000,C 90.000,E1 276.486} C_DIS
LIN {X 0.220,Y -626.713,Z 466.330,A 0.000,B 0.000,C 90.000,E1 275.454} C_DIS
LIN {X 0.136,Y -625.398,Z 466.323,A 0.000,B 0.000,C 90.000,E1 274.188} C_DIS
LIN {X -0.061,Y -624.460,Z 466.319,A 0.000,B 0.000,C 90.000,E1 273.440} C_DIS
LIN {X 0.061,Y -623.011,Z 466.313,A 0.000,B 0.000,C 90.000,E1 272.407} C_DIS
LIN {X 0.160,Y -621.358,Z 466.308,A 0.000,B 0.000,C 90.000,E1 271.375} C_DIS
LIN {X 0.238,Y -618.593,Z 466.299,A 0.000,B 0.000,C 90.000,E1 269.828} C_DIS
LIN {X -0.050,Y -616.128,Z 466.292,A 0.000,B 0.000,C 90.000,E1 268.568} C_DIS
LIN {X 0.268,Y -614.506,Z 466.288,A 0.000,B 0.000,C 90.000,E1 267.764} C_DIS
LIN {X -0.067,Y -611.736,Z 466.281,A 0.000,B 0.000,C 90.000,E1 266.502} C_DIS
LIN {X -0.121,Y -609.387,Z 466.275,A 0.000,B 0.000,C 90.000,E1 265.469} C_DIS
LIN {X 0.103,Y -606.306,Z 466.268,A 0.000,B 0.000,C 90.000,E1 264.147} C_DIS
LIN {X -0.029,Y -602.517,Z 466.259,A 0.000,B 0.000,C 90.000,E1 262.591} C_DIS
LIN {X -0.078,Y -599.899,Z 466.253,A 0.000,B 0.000,C 90.000,E1 261.546} C_DIS
LIN {X 0.139,Y -596.560,Z 466.246,A 0.000,B 0.000,C 90.000,E1 260.208} C_DIS
LIN {X 0.015,Y -593.756,Z 466.240,A 0.000,B 0.000,C 90.000,E1 259.162} C_DIS
LIN {X -0.155,Y -590.875,Z 466.234,A 0.000,B 0.000,C 90.000,E1 258.117} C_DIS
LIN {X -0.175,Y -586.423,Z 466.225,A 0.000,B 0.000,C 90.000,E1 256.520} C_DIS
LIN {X -0.039,Y -581.175,Z 466.215,A 0.000,B 0.000,C 90.000,E1 254.629} C_DIS
LIN {X 0.089,Y -577.259,Z 466.207,A 0.000,B 0.000,C 90.000,E1 253.268} C_DIS
LIN {X 0.117,Y -574.087,Z 466.201,A 0.000,B 0.000,C 90.000,E1 252.181} C_DIS
LIN {X -0.269,Y -569.988,Z 466.194,A 0.000,B 0.000,C 90.000,E1 250.859} C_DIS
LIN {X 0.191,Y -565.720,Z 466.186,A 0.000,B 0.000,C 90.000,E1 249.444} C_DIS
LIN {X -0.153,Y -561.296,Z 466.178,A 0.000,B 0.000,C 90.000,E1 248.103} C_DIS
LIN {X 0.059,Y -557.562,Z 466.172,A 0.000,B 0.000,C 90.000,E1 246.975} C_DIS
LIN {X -0.226,Y -552.703,Z 466.164,A 0.000,B 0.000,C 90.000,E1 245.613} C_DIS
LIN {X -0.138,Y -547.665,Z 466.157,A 0.000,B 0.000,C 90.000,E1 244.204} C_DIS
LIN {X -0.132,Y -542.647,Z 466.149,A 0.000,B 0.000,C 90.000,E1 242.794} C_DIS
LIN {X -0.039,Y -535.648,Z 466.138,A 0.000,B 0.000,C 90.000,E1 240.795} C_DIS
LIN {X -0.044,Y -529.577,Z 466.128,A 0.000,B 0.000,C 90.000,E1 239.076} C_DIS
LIN {X 0.002,Y -521.659,Z 466.115,A 0.000,B 0.000,C 90.000,E1 236.755} C_DIS
LIN {X -0.061,Y -517.700,Z 466.109,A 0.000,B 0.000,C 90.000,E1 235.595} C_DIS
LIN {X 0.176,Y -514.619,Z 466.104,A 0.000,B 0.000,C 90.000,E1 234.689} C_DIS
LIN {X 0.032,Y -507.335,Z 466.092,A 0.000,B 0.000,C 90.000,E1 232.637} C_DIS
LIN {X -0.316,Y -498.844,Z 466.078,A 0.000,B 0.000,C 90.000,E1 229.989} C_DIS
LIN {X -0.164,Y -493.456,Z 466.068,A 0.000,B 0.000,C 90.000,E1 228.162} C_DIS
LIN {X -0.340,Y -487.435,Z 466.056,A 0.000,B 0.000,C 90.000,E1 226.053} C_DIS
LIN {X -0.133,Y -482.412,Z 466.045,A 0.000,B 0.000,C 90.000,E1 224.190} C_DIS
LIN {X 0.196,Y -475.948,Z 466.032,A 0.000,B 0.000,C 90.000,E1 221.676} C_DIS
LIN {X -0.023,Y -470.698,Z 466.020,A 0.000,B 0.000,C 90.000,E1 219.519} C_DIS
LIN {X -0.006,Y -465.732,Z 466.007,A 0.000,B 0.000,C 90.000,E1 217.317} C_DIS
LIN {X -0.040,Y -461.051,Z 465.995,A 0.000,B 0.000,C 90.000,E1 215.105} C_DIS
LIN {X 0.015,Y -455.912,Z 465.981,A 0.000,B 0.000,C 90.000,E1 212.546} C_DIS
LIN {X 0.240,Y -452.207,Z 465.970,A 0.000,B 0.000,C 90.000,E1 210.590} C_DIS
LIN {X -0.020,Y -449.826,Z 465.963,A 0.000,B 0.000,C 90.000,E1 209.333} C_DIS
LIN {X 0.066,Y -445.574,Z 465.950,A 0.000,B 0.000,C 90.000,E1 207.052} C_DIS
LIN {X 0.139,Y -442.441,Z 465.941,A 0.000,B 0.000,C 90.000,E1 205.412} C_DIS
LIN {X 0.158,Y -439.273,Z 465.932,A 0.000,B 0.000,C 90.000,E1 203.770} C_DIS
LIN {X 0.000,Y -434.310,Z 465.918,A 0.000,B 0.000,C 90.000,E1 201.153} C_DIS
LIN {X 0.033,Y -429.632,Z 465.903,A 0.000,B 0.000,C 90.000,E1 198.489} C_DIS
LIN {X 0.130,Y -425.835,Z 465.890,A 0.000,B 0.000,C 90.000,E1 196.134} C_DIS
LIN {X 0.175,Y -422.459,Z 465.877,A 0.000,B 0.000,C 90.000,E1 193.772} C_DIS
LIN {X 0.037,Y -419.295,Z 465.864,A 0.000,B 0.000,C 90.000,E1 191.422} C_DIS
LIN {X 0.019,Y -417.268,Z 465.854,A 0.000,B 0.000,C 90.000,E1 189.726} C_DIS
LIN {X -0.084,Y -414.535,Z 465.841,A 0.000,B 0.000,C 90.000,E1 187.352} C_DIS
LIN {X 0.055,Y -412.012,Z 465.828,A 0.000,B 0.000,C 90.000,E1 184.935} C_DIS
LIN {X 0.078,Y -409.248,Z 465.810,A 0.000,B 0.000,C 90.000,E1 181.835} C_DIS
LIN {X -0.013,Y -407.324,Z 465.795,A 0.000,B 0.000,C 90.000,E1 179.083} C_DIS
LIN {X -0.175,Y -405.941,Z 465.778,A 0.000,B 0.000,C 90.000,E1 175.988} C_DIS
LIN {X 0.119,Y -405.329,Z 465.753,A 0.000,B 0.000,C 90.000,E1 171.432} C_DIS
LIN {X -0.215,Y -405.822,Z 465.737,A 0.000,B 0.000,C 90.000,E1 168.701} C_DIS
LIN {X -0.175,Y -407.349,Z 465.718,A 0.000,B 0.000,C 90.000,E1 165.227} C_DIS
LIN {X 0.106,Y -410.136,Z 465.695,A 0.000,B 0.000,C 90.000,E1 161.040} C_DIS
LIN {X -0.086,Y -413.802,Z 465.674,A 0.000,B 0.000,C 90.000,E1 157.283} C_DIS
LIN {X -0.015,Y -416.936,Z 465.659,A 0.000,B 0.000,C 90.000,E1 154.537} C_DIS
LIN {X -0.054,Y -420.279,Z 465.643,A 0.000,B 0.000,C 90.000,E1 151.820} C_DIS
LIN {X -0.066,Y -422.468,Z 465.634,A 0.000,B 0.000,C 90.000,E1 150.127} C_DIS
LIN {X 0.126,Y -425.592,Z 465.621,A 0.000,B 0.000,C 90.000,E1 147.740} C_DIS
LIN {X -0.090,Y -428.366,Z 465.610,A 0.000,B 0.000,C 90.000,E1 145.754} C_DIS
LIN {X 0.148,Y -432.222,Z 465.595,A 0.000,B 0.000,C 90.000,E1 143.050} C_DIS
LIN {X 0.165,Y -435.696,Z 465.582,A 0.000,B 0.000,C 90.000,E1 140.723} C_DIS
LIN {X -0.300,Y -437.728,Z 465.575,A 0.000,B 0.000,C 90.000,E1 139.461} C_DIS
LIN {X 0.169,Y -439.776,Z 465.567,A 0.000,B 0.000,C 90.000,E1 138.081} C_DIS
LIN {X 0.082,Y -441.165,Z 465.562,A 0.000,B 0.000,C 90.000,E1 137.106} C_DIS
LIN {X -0.041,Y -442.996,Z 465.555,A 0.000,B 0.000,C 90.000,E1 135.810} C_DIS
LIN {X -0.130,Y -444.402,Z 465.547,A 0.000,B 0.000,C 90.000,E1 134.514} C_DIS
LIN {X 0.123,Y -445.454,Z 465.540,A 0.000,B 0.000,C 90.000,E1 133.176} C_DIS
LIN {X -0.239,Y -446.145,Z 465.533,A 0.000,B 0.000,C 90.000,E1 131.919} C_DIS
LIN {X 0.047,Y -446.350,Z 465.527,A 0.000,B 0.000,C 90.000,E1 130.906} C_DIS
LIN {X 0.061,Y -446.276,Z 465.524,A 0.000,B 0.000,C 90.000,E1 130.253} C_DIS
LIN {X -0.265,Y -445.989,Z 465.520,A 0.000,B 0.000,C 90.000,E1 129.644} C_DIS
LIN {X 0.073,Y -445.346,Z 465.515,A 0.000,B 0.000,C 90.000,E1 128.624} C_DIS
LIN {X 0.052,Y -444.348,Z 465.509,A 0.000,B 0.000,C 90.000,E1 127.649} C_DIS
LIN {X -0.213,Y -442.575,Z 465.502,A 0.000,B 0.000,C 90.000,E1 126.377} C_DIS
LIN {X 0.134,Y -441.518,Z 465.498,A 0.000,B 0.000,C 90.000,E1 125.678} C_DIS
LIN {X -0.171,Y -438.964,Z 465.491,A 0.000,B 0.000,C 90.000,E1 124.405} C_DIS
LIN {X 0.178,Y -436.874,Z 465.486,A 0.000,B 0.000,C 90.000,E1 123.372} C_DIS
LIN {X -0.060,Y -433.020,Z 465.476,A 0.000,B 0.000,C 90.000,E1 121.750} C_DIS
LIN {X -0.005,Y -430.071,Z 465.470,A 0.000,B 0.000,C 90.000,E1 120.512} C_DIS
LIN {X -0.043,Y -430.087,Z 465.470,A 0.000,B 0.000,C 90.000,E1 120.512} C_DIS
LIN {X -0.002,Y -431.242,Z 465.467,A 0.000,B 0.000,C 90.000,E1 120.079} C_DIS
LIN {X -0.037,Y -440.376,Z 465.447,A 0.000,B 0.000,C 90.000,E1 116.437} C_DIS
LIN {X -0.280,Y -444.212,Z 465.440,A 0.000,B 0.000,C 90.000,E1 115.155} C_DIS
LIN {X 0.164,Y -445.084,Z 465.438,A 0.000,B 0.000,C 90.000,E1 114.771} C_DIS
LIN {X -0.152,Y -454.246,Z 465.416,A 0.000,B 0.000,C 90.000,E1 110.918} C_DIS
LIN {X -0.036,Y -456.910,Z 465.411,A 0.000,B 0.000,C 90.000,E1 109.939} C_DIS
LIN {X -0.134,Y -457.621,Z 465.409,A 0.000,B 0.000,C 90.000,E1 109.631} C_DIS
LIN {X -0.048,Y -466.341,Z 465.386,A 0.000,B 0.000,C 90.000,E1 105.481} C_DIS
LIN {X 0.126,Y -467.875,Z 465.383,A 0.000,B 0.000,C 90.000,E1 104.828} C_DIS
LIN {X 0.155,Y -475.436,Z 465.358,A 0.000,B 0.000,C 90.000,E1 100.433} C_DIS
LIN {X -0.008,Y -476.087,Z 465.356,A 0.000,B 0.000,C 90.000,E1 100.141} C_DIS
LIN {X -0.029,Y -477.429,Z 465.349,A 0.000,B 0.000,C 90.000,E1 98.859} C_DIS
LIN {X -0.068,Y -541.120,Z 465.349,A 0.000,B 0.000,C 90.000,E1 98.859} C_DIS
LIN {X 0.162,Y -547.218,Z 465.349,A 0.000,B 0.000,C 90.000,E1 98.803} C_DIS
LIN {X -0.119,Y -554.236,Z 465.349,A 0.000,B 0.000,C 90.000,E1 98.746} C_DIS
LIN {X 0.003,Y -560.184,Z 465.348,A 0.000,B 0.000,C 90.000,E1 98.624} C_DIS
LIN {X 0.176,Y -568.677,Z 465.347,A 0.000,B 0.000,C 90.000,E1 98.398} C_DIS
LIN {X 0.067,Y -575.308,Z 465.346,A 0.000,B 0.000,C 90.000,E1 98.219} C_DIS
LIN {X 0.142,Y -581.851,Z 465.345,A 0.000,B 0.000,C 90.000,E1 97.992} C_DIS
LIN {X 0.196,Y -591.557,Z 465.342,A 0.000,B 0.000,C 90.000,E1 97.587} C_DIS
LIN {X 0.193,Y -597.769,Z 465.341,A 0.000,B 0.000,C 90.000,E1 97.296} C_DIS
LIN {X -0.223,Y -603.695,Z 465.339,A 0.000,B 0.000,C 90.000,E1 97.004} C_DIS
LIN {X -0.023,Y -609.482,Z 465.337,A 0.000,B 0.000,C 90.000,E1 96.606} C_DIS
LIN {X -0.042,Y -616.517,Z 465.334,A 0.000,B 0.000,C 90.000,E1 96.087} C_DIS
LIN {X -0.143,Y -622.885,Z 465.331,A 0.000,B 0.000,C 90.000,E1 95.511} C_DIS
LIN {X 0.237,Y -625.674,Z 465.329,A 0.000,B 0.000,C 90.000,E1 95.106} C_DIS
LIN {X -0.095,Y -628.892,Z 465.327,A 0.000,B 0.000,C 90.000,E1 94.821} C_DIS
LIN {X 0.221,Y -635.335,Z 465.321,A 0.000,B 0.000,C 90.000,E1 93.784} C_DIS
LIN {X -0.040,Y -636.584,Z 465.320,A 0.000,B 0.000,C 90.000,E1 93.555} C_DIS
LIN {X -0.297,Y -637.546,Z 465.318,A 0.000,B 0.000,C 90.000,E1 93.326} C_DIS
LIN {X 0.120,Y -638.725,Z 465.317,A 0.000,B 0.000,C 90.000,E1 93.037} C_DIS
LIN {X 0.260,Y -640.747,Z 465.314,A 0.000,B 0.000,C 90.000,E1 92.522} C_DIS
LIN {X 0.017,Y -641.530,Z 465.313,A 0.000,B 0.000,C 90.000,E1 92.293} C_DIS
LIN {X 0.204,Y -642.761,Z 465.310,A 0.000,B 0.000,C 90.000,E1 91.776} C_DIS
LIN {X 0.145,Y -643.829,Z 465.306,A 0.000,B 0.000,C 90.000,E1 91.031} C_DIS
LIN {X -0.315,Y -644.179,Z 465.303,A 0.000,B 0.000,C 90.000,E1 90.573} C_DIS
LIN {X -0.127,Y -644.186,Z 465.300,A 0.000,B 0.000,C 90.000,E1 90.057} C_DIS
LIN {X 0.061,Y -643.788,Z 465.298,A 0.000,B 0.000,C 90.000,E1 89.542} C_DIS
LIN {X 0.016,Y -642.561,Z 465.293,A 0.000,B 0.000,C 90.000,E1 88.797} C_DIS
LIN {X 0.191,Y -641.378,Z 465.291,A 0.000,B 0.000,C 90.000,E1 88.282} C_DIS
LIN {X -0.024,Y -640.620,Z 465.289,A 0.000,B 0.000,C 90.000,E1 88.051} C_DIS
LIN {X -0.261,Y -639.706,Z 465.288,A 0.000,B 0.000,C 90.000,E1 87.822} C_DIS
LIN {X 0.018,Y -637.900,Z 465.286,A 0.000,B 0.000,C 90.000,E1 87.421} C_DIS
LIN {X -0.066,Y -633.980,Z 465.282,A 0.000,B 0.000,C 90.000,E1 86.674} C_DIS
LIN {X 0.306,Y -628.209,Z 465.277,A 0.000,B 0.000,C 90.000,E1 85.755} C_DIS
LIN {X 0.125,Y -622.370,Z 465.272,A 0.000,B 0.000,C 90.000,E1 85.008} C_DIS
LIN {X 0.041,Y -616.571,Z 465.269,A 0.000,B 0.000,C 90.000,E1 84.375} C_DIS
LIN {X 0.088,Y -610.093,Z 465.265,A 0.000,B 0.000,C 90.000,E1 83.742} C_DIS
LIN {X 0.281,Y -604.698,Z 465.263,A 0.000,B 0.000,C 90.000,E1 83.280} C_DIS
LIN {X -0.097,Y -598.597,Z 465.260,A 0.000,B 0.000,C 90.000,E1 82.875} C_DIS
LIN {X -0.233,Y -589.038,Z 465.257,A 0.000,B 0.000,C 90.000,E1 82.299} C_DIS
LIN {X 0.218,Y -585.619,Z 465.256,A 0.000,B 0.000,C 90.000,E1 82.064} C_DIS
LIN {X -0.015,Y -580.515,Z 465.255,A 0.000,B 0.000,C 90.000,E1 81.837} C_DIS
LIN {X 0.254,Y -576.777,Z 465.254,A 0.000,B 0.000,C 90.000,E1 81.659} C_DIS
LIN {X 0.025,Y -572.760,Z 465.253,A 0.000,B 0.000,C 90.000,E1 81.546} C_DIS
LIN {X 0.202,Y -567.386,Z 465.252,A 0.000,B 0.000,C 90.000,E1 81.376} C_DIS
LIN {X -0.188,Y -561.464,Z 465.252,A 0.000,B 0.000,C 90.000,E1 81.310} C_DIS
LIN {X 0.235,Y -554.893,Z 465.251,A 0.000,B 0.000,C 90.000,E1 81.197} C_DIS
LIN {X 0.179,Y -550.297,Z 465.251,A 0.000,B 0.000,C 90.000,E1 81.197} C_DIS
LIN {X 0.110,Y -484.263,Z 465.251,A 0.000,B 0.000,C 90.000,E1 81.197} C_DIS
LIN {X -0.176,Y -480.529,Z 465.227,A 0.000,B 0.000,C 90.000,E1 76.881} C_DIS
LIN {X 0.188,Y -474.279,Z 465.201,A 0.000,B 0.000,C 90.000,E1 72.181} C_DIS
LIN {X 0.156,Y -473.835,Z 465.199,A 0.000,B 0.000,C 90.000,E1 71.873} C_DIS
LIN {X 0.116,Y -466.247,Z 465.175,A 0.000,B 0.000,C 90.000,E1 67.486} C_DIS
LIN {X 0.058,Y -465.818,Z 465.173,A 0.000,B 0.000,C 90.000,E1 67.177} C_DIS
LIN {X -0.002,Y -465.218,Z 465.172,A 0.000,B 0.000,C 90.000,E1 66.869} C_DIS
LIN {X 0.039,Y -457.443,Z 465.151,A 0.000,B 0.000,C 90.000,E1 63.076} C_DIS
LIN {X 0.000,Y -457.462,Z 465.150,A 0.000,B 0.000,C 90.000,E1 63.076} C_DIS
LIN {X 0.098,Y -465.822,Z 465.143,A 0.000,B 0.000,C 90.000,E1 61.769} C_DIS
LIN {X -0.073,Y -470.779,Z 465.139,A 0.000,B 0.000,C 90.000,E1 61.001} C_DIS
LIN {X 0.030,Y -476.486,Z 465.134,A 0.000,B 0.000,C 90.000,E1 60.049} C_DIS
LIN {X -0.054,Y -480.747,Z 465.129,A 0.000,B 0.000,C 90.000,E1 59.282} C_DIS
LIN {X -0.046,Y -483.873,Z 465.126,A 0.000,B 0.000,C 90.000,E1 58.663} C_DIS
LIN {X 0.183,Y -487.214,Z 465.122,A 0.000,B 0.000,C 90.000,E1 57.867} C_DIS
LIN {X -0.213,Y -489.002,Z 465.119,A 0.000,B 0.000,C 90.000,E1 57.454} C_DIS
LIN {X 0.105,Y -492.049,Z 465.114,A 0.000,B 0.000,C 90.000,E1 56.501} C_DIS
LIN {X 0.203,Y -493.671,Z 465.111,A 0.000,B 0.000,C 90.000,E1 55.881} C_DIS
LIN {X 0.168,Y -495.571,Z 465.106,A 0.000,B 0.000,C 90.000,E1 54.975} C_DIS
LIN {X 0.152,Y -496.912,Z 465.101,A 0.000,B 0.000,C 90.000,E1 54.069} C_DIS
LIN {X -0.120,Y -497.650,Z 465.097,A 0.000,B 0.000,C 90.000,E1 53.497} C_DIS
LIN {X 0.181,Y -498.389,Z 465.092,A 0.000,B 0.000,C 90.000,E1 52.557} C_DIS
LIN {X 0.102,Y -498.880,Z 465.087,A 0.000,B 0.000,C 90.000,E1 51.662} C_DIS
LIN {X -0.094,Y -499.130,Z 465.080,A 0.000,B 0.000,C 90.000,E1 50.481} C_DIS
LIN {X 0.031,Y -499.201,Z 465.077,A 0.000,B 0.000,C 90.000,E1 49.865} C_DIS
LIN {X -0.225,Y -498.982,Z 465.070,A 0.000,B 0.000,C 90.000,E1 48.690} C_DIS
LIN {X -0.104,Y -498.618,Z 465.064,A 0.000,B 0.000,C 90.000,E1 47.472} C_DIS
LIN {X -0.161,Y -498.004,Z 465.055,A 0.000,B 0.000,C 90.000,E1 45.972} C_DIS
LIN {X -0.077,Y -497.355,Z 465.049,A 0.000,B 0.000,C 90.000,E1 44.757} C_DIS
LIN {X 0.184,Y -496.419,Z 465.040,A 0.000,B 0.000,C 90.000,E1 43.218} C_DIS
LIN {X -0.106,Y -495.535,Z 465.034,A 0.000,B 0.000,C 90.000,E1 42.043} C_DIS
LIN {X -0.017,Y -494.124,Z 465.023,A 0.000,B 0.000,C 90.000,E1 40.216} C_DIS
LIN {X -0.055,Y -492.845,Z 465.015,A 0.000,B 0.000,C 90.000,E1 38.705} C_DIS
LIN {X -0.044,Y -491.858,Z 465.008,A 0.000,B 0.000,C 90.000,E1 37.488} C_DIS
LIN {X -0.017,Y -490.505,Z 465.000,A 0.000,B 0.000,C 90.000,E1 35.964} C_DIS
LIN {X 0.038,Y -489.257,Z 464.993,A 0.000,B 0.000,C 90.000,E1 34.739} C_DIS
LIN {X 0.190,Y -488.002,Z 464.986,A 0.000,B 0.000,C 90.000,E1 33.499} C_DIS
LIN {X 0.062,Y -486.600,Z 464.979,A 0.000,B 0.000,C 90.000,E1 32.291} C_DIS
LIN {X 0.170,Y -485.168,Z 464.973,A 0.000,B 0.000,C 90.000,E1 31.052} C_DIS
LIN {X -0.247,Y -483.639,Z 464.966,A 0.000,B 0.000,C 90.000,E1 29.873} C_DIS
LIN {X 0.175,Y -481.394,Z 464.956,A 0.000,B 0.000,C 90.000,E1 27.975} C_DIS
LIN {X 0.043,Y -478.201,Z 464.940,A 0.000,B 0.000,C 90.000,E1 25.207} C_DIS
LIN {X 0.051,Y -475.472,Z 464.923,A 0.000,B 0.000,C 90.000,E1 22.099} C_DIS
LIN {X -0.124,Y -473.977,Z 464.911,A 0.000,B 0.000,C 90.000,E1 19.939} C_DIS
LIN {X 0.191,Y -472.483,Z 464.897,A 0.000,B 0.000,C 90.000,E1 17.402} C_DIS
LIN {X -0.092,Y -471.091,Z 464.885,A 0.000,B 0.000,C 90.000,E1 15.245} C_DIS
LIN {X -0.205,Y -469.868,Z 464.872,A 0.000,B 0.000,C 90.000,E1 13.063} C_DIS
LIN {X 0.011,Y -469.071,Z 464.860,A 0.000,B 0.000,C 90.000,E1 10.838} C_DIS
LIN {X -0.145,Y -468.574,Z 464.846,A 0.000,B 0.000,C 90.000,E1 8.341} C_DIS
LIN {X -0.132,Y -468.655,Z 464.827,A 0.000,B 0.000,C 90.000,E1 4.878} C_DIS
LIN {X 0.230,Y -469.973,Z 464.808,A 0.000,B 0.000,C 90.000,E1 1.375} C_DIS
LIN {X 0.009,Y -472.274,Z 464.790,A 0.000,B 0.000,C 90.000,E1 358.224} C_DIS
LIN {X 0.222,Y -474.803,Z 464.776,A 0.000,B 0.000,C 90.000,E1 355.698} C_DIS
LIN {X 0.090,Y -477.780,Z 464.762,A 0.000,B 0.000,C 90.000,E1 353.223} C_DIS
LIN {X -0.168,Y -480.755,Z 464.750,A 0.000,B 0.000,C 90.000,E1 351.084} C_DIS
LIN {X 0.077,Y -483.143,Z 464.742,A 0.000,B 0.000,C 90.000,E1 349.511} C_DIS
LIN {X -0.008,Y -491.068,Z 464.718,A 0.000,B 0.000,C 90.000,E1 345.227} C_DIS
LIN {X 0.045,Y -497.142,Z 464.703,A 0.000,B 0.000,C 90.000,E1 342.489} C_DIS
LIN {X 0.217,Y -503.048,Z 464.689,A 0.000,B 0.000,C 90.000,E1 340.061} C_DIS
LIN {X 0.176,Y -508.317,Z 464.678,A 0.000,B 0.000,C 90.000,E1 337.975} C_DIS
LIN {X -0.126,Y -512.771,Z 464.668,A 0.000,B 0.000,C 90.000,E1 336.230} C_DIS
LIN {X -0.123,Y -515.710,Z 464.661,A 0.000,B 0.000,C 90.000,E1 335.049} C_DIS
LIN {X 0.135,Y -518.597,Z 464.655,A 0.000,B 0.000,C 90.000,E1 333.845} C_DIS
LIN {X -0.115,Y -522.233,Z 464.647,A 0.000,B 0.000,C 90.000,E1 332.410} C_DIS
LIN {X -0.147,Y -526.579,Z 464.637,A 0.000,B 0.000,C 90.000,E1 330.667} C_DIS
LIN {X -0.020,Y -531.041,Z 464.627,A 0.000,B 0.000,C 90.000,E1 328.918} C_DIS
LIN {X 0.215,Y -535.519,Z 464.618,A 0.000,B 0.000,C 90.000,E1 327.168} C_DIS
LIN {X 0.088,Y -540.015,Z 464.608,A 0.000,B 0.000,C 90.000,E1 325.468} C_DIS
LIN {X -0.060,Y -545.360,Z 464.597,A 0.000,B 0.000,C 90.000,E1 323.497} C_DIS
LIN {X -0.237,Y -550.023,Z 464.588,A 0.000,B 0.000,C 90.000,E1 321.823} C_DIS
LIN {X 0.104,Y -555.378,Z 464.577,A 0.000,B 0.000,C 90.000,E1 319.828} C_DIS
LIN {X 0.150,Y -560.772,Z 464.566,A 0.000,B 0.000,C 90.000,E1 317.877} C_DIS
LIN {X 0.033,Y -563.825,Z 464.560,A 0.000,B 0.000,C 90.000,E1 316.782} C_DIS
LIN {X -0.273,Y -568.378,Z 464.551,A 0.000,B 0.000,C 90.000,E1 315.162} C_DIS
LIN {X 0.029,Y -573.593,Z 464.540,A 0.000,B 0.000,C 90.000,E1 313.218} C_DIS
LIN {X -0.052,Y -578.052,Z 464.531,A 0.000,B 0.000,C 90.000,E1 311.595} C_DIS
LIN {X 0.022,Y -582.382,Z 464.522,A 0.000,B 0.000,C 90.000,E1 309.967} C_DIS
LIN {X 0.011,Y -586.082,Z 464.515,A 0.000,B 0.000,C 90.000,E1 308.624} C_DIS
LIN {X -0.103,Y -590.319,Z 464.506,A 0.000,B 0.000,C 90.000,E1 307.030} C_DIS
LIN {X -0.140,Y -594.500,Z 464.497,A 0.000,B 0.000,C 90.000,E1 305.438} C_DIS
LIN {X -0.194,Y -597.921,Z 464.490,A 0.000,B 0.000,C 90.000,E1 304.119} C_DIS
LIN {X -0.279,Y -601.702,Z 464.481,A 0.000,B 0.000,C 90.000,E1 302.546} C_DIS
LIN {X 0.221,Y -605.312,Z 464.472,A 0.000,B 0.000,C 90.000,E1 300.924} C_DIS
LIN {X 0.288,Y -607.568,Z 464.466,A 0.000,B 0.000,C 90.000,E1 299.873} C_DIS
LIN {X -0.189,Y -610.139,Z 464.459,A 0.000,B 0.000,C 90.000,E1 298.615} C_DIS
LIN {X -0.195,Y -614.130,Z 464.447,A 0.000,B 0.000,C 90.000,E1 296.539} C_DIS
LIN {X 0.254,Y -615.947,Z 464.442,A 0.000,B 0.000,C 90.000,E1 295.463} C_DIS
LIN {X -0.101,Y -617.946,Z 464.434,A 0.000,B 0.000,C 90.000,E1 294.207} C_DIS
LIN {X 0.131,Y -620.164,Z 464.426,A 0.000,B 0.000,C 90.000,E1 292.642} C_DIS
LIN {X 0.180,Y -621.848,Z 464.419,A 0.000,B 0.000,C 90.000,E1 291.354} C_DIS
LIN {X -0.094,Y -623.079,Z 464.413,A 0.000,B 0.000,C 90.000,E1 290.355} C_DIS
LIN {X 0.009,Y -624.331,Z 464.407,A 0.000,B 0.000,C 90.000,E1 289.322} C_DIS
LIN {X 0.276,Y -626.208,Z 464.397,A 0.000,B 0.000,C 90.000,E1 287.511} C_DIS
LIN {X 0.025,Y -627.427,Z 464.390,A 0.000,B 0.000,C 90.000,E1 286.260} C_DIS
LIN {X 0.207,Y -628.566,Z 464.382,A 0.000,B 0.000,C 90.000,E1 284.717} C_DIS
LIN {X 0.037,Y -629.238,Z 464.376,A 0.000,B 0.000,C 90.000,E1 283.716} C_DIS
LIN {X -0.316,Y -629.856,Z 464.369,A 0.000,B 0.000,C 90.000,E1 282.479} C_DIS
LIN {X -0.049,Y -630.302,Z 464.362,A 0.000,B 0.000,C 90.000,E1 281.186} C_DIS
LIN {X -0.326,Y -630.481,Z 464.357,A 0.000,B 0.000,C 90.000,E1 280.197} C_DIS
LIN {X -0.178,Y -630.468,Z 464.349,A 0.000,B 0.000,C 90.000,E1 278.916} C_DIS
LIN {X -0.130,Y -630.184,Z 464.342,A 0.000,B 0.000,C 90.000,E1 277.644} C_DIS
LIN {X 0.125,Y -629.662,Z 464.337,A 0.000,B 0.000,C 90.000,E1 276.606} C_DIS
LIN {X 0.151,Y -628.754,Z 464.330,A 0.000,B 0.000,C 90.000,E1 275.334} C_DIS
LIN {X -0.301,Y -627.679,Z 464.324,A 0.000,B 0.000,C 90.000,E1 274.359} C_DIS
LIN {X 0.150,Y -626.734,Z 464.320,A 0.000,B 0.000,C 90.000,E1 273.555} C_DIS
LIN {X 0.018,Y -624.874,Z 464.313,A 0.000,B 0.000,C 90.000,E1 272.293} C_DIS
LIN {X 0.141,Y -623.154,Z 464.307,A 0.000,B 0.000,C 90.000,E1 271.260} C_DIS
LIN {X -0.069,Y -620.793,Z 464.300,A 0.000,B 0.000,C 90.000,E1 270.000} C_DIS
LIN {X 0.300,Y -618.360,Z 464.293,A 0.000,B 0.000,C 90.000,E1 268.682} C_DIS
LIN {X -0.284,Y -616.143,Z 464.287,A 0.000,B 0.000,C 90.000,E1 267.707} C_DIS
LIN {X 0.022,Y -613.323,Z 464.280,A 0.000,B 0.000,C 90.000,E1 266.388} C_DIS
LIN {X -0.013,Y -610.895,Z 464.274,A 0.000,B 0.000,C 90.000,E1 265.355} C_DIS
LIN {X -0.029,Y -608.406,Z 464.268,A 0.000,B 0.000,C 90.000,E1 264.318} C_DIS
LIN {X -0.112,Y -604.579,Z 464.260,A 0.000,B 0.000,C 90.000,E1 262.761} C_DIS
LIN {X 0.093,Y -601.270,Z 464.253,A 0.000,B 0.000,C 90.000,E1 261.432} C_DIS
LIN {X 0.037,Y -597.200,Z 464.244,A 0.000,B 0.000,C 90.000,E1 259.859} C_DIS
LIN {X 0.204,Y -593.606,Z 464.236,A 0.000,B 0.000,C 90.000,E1 258.522} C_DIS
LIN {X 0.108,Y -589.097,Z 464.228,A 0.000,B 0.000,C 90.000,E1 256.937} C_DIS
LIN {X -0.329,Y -585.275,Z 464.220,A 0.000,B 0.000,C 90.000,E1 255.644} C_DIS
LIN {X 0.207,Y -582.243,Z 464.214,A 0.000,B 0.000,C 90.000,E1 254.519} C_DIS
LIN {X -0.043,Y -578.306,Z 464.207,A 0.000,B 0.000,C 90.000,E1 253.196} C_DIS
LIN {X 0.197,Y -574.226,Z 464.199,A 0.000,B 0.000,C 90.000,E1 251.819} C_DIS
LIN {X 0.187,Y -570.902,Z 464.193,A 0.000,B 0.000,C 90.000,E1 250.732} C_DIS
LIN {X -0.067,Y -566.591,Z 464.186,A 0.000,B 0.000,C 90.000,E1 249.390} C_DIS
LIN {X -0.189,Y -562.159,Z 464.178,A 0.000,B 0.000,C 90.000,E1 248.028} C_DIS
LIN {X -0.177,Y -558.364,Z 464.172,A 0.000,B 0.000,C 90.000,E1 246.922} C_DIS
LIN {X -0.221,Y -553.463,Z 464.164,A 0.000,B 0.000,C 90.000,E1 245.537} C_DIS
LIN {X 0.140,Y -548.400,Z 464.156,A 0.000,B 0.000,C 90.000,E1 244.101} C_DIS
LIN {X 0.144,Y -543.311,Z 464.148,A 0.000,B 0.000,C 90.000,E1 242.692} C_DIS
LIN {X 0.027,Y -536.273,Z 464.137,A 0.000,B 0.000,C 90.000,E1 240.717} C_DIS
LIN {X 0.042,Y -530.194,Z 464.128,A 0.000,B 0.000,C 90.000,E1 238.997} C_DIS
LIN {X -0.177,Y -522.231,Z 464.115,A 0.000,B 0.000,C 90.000,E1 236.707} C_DIS
LIN {X 0.001,Y -517.257,Z 464.107,A 0.000,B 0.000,C 90.000,E1 235.229} C_DIS
LIN {X 0.018,Y -510.997,Z 464.097,A 0.000,B 0.000,C 90.000,E1 233.463} C_DIS
LIN {X -0.155,Y -499.418,Z 464.077,A 0.000,B 0.000,C 90.000,E1 229.908} C_DIS
LIN {X 0.010,Y -494.052,Z 464.067,A 0.000,B 0.000,C 90.000,E1 228.081} C_DIS
LIN {X -0.151,Y -488.023,Z 464.055,A 0.000,B 0.000,C 90.000,E1 225.972} C_DIS
LIN {X 0.204,Y -482.162,Z 464.043,A 0.000,B 0.000,C 90.000,E1 223.785} C_DIS
LIN {X -0.262,Y -476.545,Z 464.031,A 0.000,B 0.000,C 90.000,E1 221.676} C_DIS
LIN {X -0.162,Y -471.286,Z 464.019,A 0.000,B 0.000,C 90.000,E1 219.483} C_DIS
LIN {X 0.092,Y -466.993,Z 464.009,A 0.000,B 0.000,C 90.000,E1 217.569} C_DIS
LIN {X -0.190,Y -462.256,Z 463.997,A 0.000,B 0.000,C 90.000,E1 215.391} C_DIS
LIN {X 0.058,Y -458.312,Z 463.986,A 0.000,B 0.000,C 90.000,E1 213.452} C_DIS
LIN {X -0.143,Y -455.200,Z 463.977,A 0.000,B 0.000,C 90.000,E1 211.878} C_DIS
LIN {X -0.068,Y -450.947,Z 463.965,A 0.000,B 0.000,C 90.000,E1 209.617} C_DIS
LIN {X 0.062,Y -446.670,Z 463.952,A 0.000,B 0.000,C 90.000,E1 207.334} C_DIS
LIN {X -0.041,Y -443.531,Z 463.943,A 0.000,B 0.000,C 90.000,E1 205.720} C_DIS
LIN {X -0.003,Y -440.366,Z 463.934,A 0.000,B 0.000,C 90.000,E1 204.079} C_DIS
LIN {X 0.040,Y -435.933,Z 463.921,A 0.000,B 0.000,C 90.000,E1 201.770} C_DIS
LIN {X -0.183,Y -432.282,Z 463.910,A 0.000,B 0.000,C 90.000,E1 199.812} C_DIS
LIN {X -0.012,Y -428.328,Z 463.897,A 0.000,B 0.000,C 90.000,E1 197.457} C_DIS
LIN {X -0.158,Y -423.246,Z 463.878,A 0.000,B 0.000,C 90.000,E1 194.120} C_DIS
LIN {X 0.133,Y -420.027,Z 463.865,A 0.000,B 0.000,C 90.000,E1 191.715} C_DIS
LIN {X 0.191,Y -417.550,Z 463.854,A 0.000,B 0.000,C 90.000,E1 189.670} C_DIS
LIN {X 0.098,Y -414.805,Z 463.841,A 0.000,B 0.000,C 90.000,E1 187.296} C_DIS
LIN {X -0.166,Y -412.285,Z 463.827,A 0.000,B 0.000,C 90.000,E1 184.935} C_DIS
LIN {X -0.129,Y -409.212,Z 463.808,A 0.000,B 0.000,C 90.000,E1 181.489} C_DIS
LIN {X 0.154,Y -407.045,Z 463.789,A 0.000,B 0.000,C 90.000,E1 177.993} C_DIS
LIN {X 0.012,Y -405.885,Z 463.772,A 0.000,B 0.000,C 90.000,E1 174.894} C_DIS
LIN {X -0.059,Y -405.616,Z 463.752,A 0.000,B 0.000,C 90.000,E1 171.432} C_DIS
LIN {X 0.094,Y -406.137,Z 463.737,A 0.000,B 0.000,C 90.000,E1 168.634} C_DIS
LIN {X 0.064,Y -407.699,Z 463.718,A 0.000,B 0.000,C 90.000,E1 165.172} C_DIS
LIN {X 0.093,Y -410.826,Z 463.693,A 0.000,B 0.000,C 90.000,E1 160.678} C_DIS
LIN {X 0.174,Y -414.226,Z 463.674,A 0.000,B 0.000,C 90.000,E1 157.230} C_DIS
LIN {X -0.123,Y -417.403,Z 463.658,A 0.000,B 0.000,C 90.000,E1 154.537} C_DIS
LIN {X -0.064,Y -419.942,Z 463.647,A 0.000,B 0.000,C 90.000,E1 152.487} C_DIS
LIN {X -0.119,Y -422.634,Z 463.636,A 0.000,B 0.000,C 90.000,E1 150.461} C_DIS
LIN {X 0.062,Y -426.252,Z 463.621,A 0.000,B 0.000,C 90.000,E1 147.740} C_DIS
LIN {X 0.102,Y -429.126,Z 463.610,A 0.000,B 0.000,C 90.000,E1 145.722} C_DIS
LIN {X 0.123,Y -433.108,Z 463.595,A 0.000,B 0.000,C 90.000,E1 143.050} C_DIS
LIN {X -0.173,Y -437.216,Z 463.580,A 0.000,B 0.000,C 90.000,E1 140.436} C_DIS
LIN {X -0.089,Y -440.389,Z 463.569,A 0.000,B 0.000,C 90.000,E1 138.447} C_DIS
LIN {X -0.197,Y -442.364,Z 463.562,A 0.000,B 0.000,C 90.000,E1 137.148} C_DIS
LIN {X 0.024,Y -444.257,Z 463.555,A 0.000,B 0.000,C 90.000,E1 135.810} C_DIS
LIN {X -0.045,Y -445.768,Z 463.547,A 0.000,B 0.000,C 90.000,E1 134.514} C_DIS
LIN {X -0.097,Y -446.908,Z 463.540,A 0.000,B 0.000,C 90.000,E1 133.218} C_DIS
LIN {X -0.110,Y -447.704,Z 463.533,A 0.000,B 0.000,C 90.000,E1 131.919} C_DIS
LIN {X 0.195,Y -447.957,Z 463.527,A 0.000,B 0.000,C 90.000,E1 130.906} C_DIS
LIN {X 0.208,Y -447.828,Z 463.522,A 0.000,B 0.000,C 90.000,E1 129.930} C_DIS
LIN {X 0.236,Y -447.482,Z 463.518,A 0.000,B 0.000,C 90.000,E1 129.277} C_DIS
LIN {X -0.085,Y -447.049,Z 463.515,A 0.000,B 0.000,C 90.000,E1 128.669} C_DIS
LIN {X -0.010,Y -446.067,Z 463.509,A 0.000,B 0.000,C 90.000,E1 127.684} C_DIS
LIN {X 0.022,Y -444.320,Z 463.502,A 0.000,B 0.000,C 90.000,E1 126.377} C_DIS
LIN {X -0.285,Y -443.880,Z 463.500,A 0.000,B 0.000,C 90.000,E1 126.091} C_DIS
LIN {X 0.061,Y -441.385,Z 463.493,A 0.000,B 0.000,C 90.000,E1 124.739} C_DIS
LIN {X -0.175,Y -439.311,Z 463.488,A 0.000,B 0.000,C 90.000,E1 123.785} C_DIS
LIN {X 0.144,Y -437.791,Z 463.484,A 0.000,B 0.000,C 90.000,E1 123.086} C_DIS
LIN {X -0.080,Y -433.874,Z 463.475,A 0.000,B 0.000,C 90.000,E1 121.465} C_DIS
LIN {X -0.080,Y -430.876,Z 463.468,A 0.000,B 0.000,C 90.000,E1 120.256} C_DIS
LIN {X -0.118,Y -430.883,Z 463.468,A 0.000,B 0.000,C 90.000,E1 120.256} C_DIS
LIN {X -0.068,Y -440.242,Z 463.447,A 0.000,B 0.000,C 90.000,E1 116.488} C_DIS
LIN {X -0.062,Y -444.989,Z 463.438,A 0.000,B 0.000,C 90.000,E1 114.847} C_DIS
LIN {X 0.215,Y -454.122,Z 463.416,A 0.000,B 0.000,C 90.000,E1 110.918} C_DIS
LIN {X -0.098,Y -456.778,Z 463.411,A 0.000,B 0.000,C 90.000,E1 109.993} C_DIS
LIN {X 0.233,Y -457.540,Z 463.409,A 0.000,B 0.000,C 90.000,E1 109.631} C_DIS
LIN {X -0.127,Y -466.230,Z 463.386,A 0.000,B 0.000,C 90.000,E1 105.536} C_DIS
LIN {X -0.077,Y -467.790,Z 463.383,A 0.000,B 0.000,C 90.000,E1 104.898} C_DIS
LIN {X -0.104,Y -475.996,Z 463.357,A 0.000,B 0.000,C 90.000,E1 100.197} C_DIS
LIN {X 0.044,Y -476.692,Z 463.353,A 0.000,B 0.000,C 90.000,E1 99.557} C_DIS
LIN {X -0.030,Y -478.018,Z 463.346,A 0.000,B 0.000,C 90.000,E1 98.341} C_DIS
LIN {X -0.080,Y -545.970,Z 463.346,A 0.000,B 0.000,C 90.000,E1 98.341} C_DIS
LIN {X -0.214,Y -550.376,Z 463.346,A 0.000,B 0.000,C 90.000,E1 98.341} C_DIS
LIN {X -0.227,Y -556.061,Z 463.346,A 0.000,B 0.000,C 90.000,E1 98.276} C_DIS
LIN {X -0.229,Y -562.570,Z 463.345,A 0.000,B 0.000,C 90.000,E1 98.163} C_DIS
LIN {X 0.038,Y -568.863,Z 463.344,A 0.000,B 0.000,C 90.000,E1 97.992} C_DIS
LIN {X 0.068,Y -575.398,Z 463.344,A 0.000,B 0.000,C 90.000,E1 97.814} C_DIS
LIN {X 0.179,Y -578.854,Z 463.343,A 0.000,B 0.000,C 90.000,E1 97.701} C_DIS
LIN {X 0.204,Y -585.249,Z 463.342,A 0.000,B 0.000,C 90.000,E1 97.473} C_DIS
LIN {X -0.114,Y -591.507,Z 463.340,A 0.000,B 0.000,C 90.000,E1 97.239} C_DIS
LIN {X -0.175,Y -597.887,Z 463.339,A 0.000,B 0.000,C 90.000,E1 96.947} C_DIS
LIN {X -0.049,Y -603.915,Z 463.337,A 0.000,B 0.000,C 90.000,E1 96.606} C_DIS
LIN {X -0.245,Y -609.715,Z 463.335,A 0.000,B 0.000,C 90.000,E1 96.258} C_DIS
LIN {X 0.303,Y -616.478,Z 463.332,A 0.000,B 0.000,C 90.000,E1 95.682} C_DIS
LIN {X 0.270,Y -621.622,Z 463.329,A 0.000,B 0.000,C 90.000,E1 95.220} C_DIS
LIN {X 0.194,Y -622.732,Z 463.329,A 0.000,B 0.000,C 90.000,E1 95.106} C_DIS
LIN {X 0.042,Y -623.653,Z 463.328,A 0.000,B 0.000,C 90.000,E1 94.992} C_DIS
LIN {X -0.110,Y -624.973,Z 463.327,A 0.000,B 0.000,C 90.000,E1 94.878} C_DIS
LIN {X 0.295,Y -628.649,Z 463.325,A 0.000,B 0.000,C 90.000,E1 94.416} C_DIS
LIN {X 0.136,Y -633.580,Z 463.320,A 0.000,B 0.000,C 90.000,E1 93.669} C_DIS
LIN {X 0.004,Y -634.331,Z 463.320,A 0.000,B 0.000,C 90.000,E1 93.555} C_DIS
LIN {X 0.019,Y -636.999,Z 463.316,A 0.000,B 0.000,C 90.000,E1 92.922} C_DIS
LIN {X 0.148,Y -638.882,Z 463.314,A 0.000,B 0.000,C 90.000,E1 92.407} C_DIS
LIN {X 0.296,Y -640.481,Z 463.311,A 0.000,B 0.000,C 90.000,E1 91.892} C_DIS
LIN {X 0.073,Y -641.015,Z 463.309,A 0.000,B 0.000,C 90.000,E1 91.661} C_DIS
LIN {X 0.235,Y -641.739,Z 463.307,A 0.000,B 0.000,C 90.000,E1 91.146} C_DIS
LIN {X -0.238,Y -642.115,Z 463.304,A 0.000,B 0.000,C 90.000,E1 90.688} C_DIS
LIN {X -0.064,Y -642.127,Z 463.301,A 0.000,B 0.000,C 90.000,E1 90.172} C_DIS
LIN {X 0.110,Y -641.793,Z 463.298,A 0.000,B 0.000,C 90.000,E1 89.656} C_DIS
LIN {X -0.124,Y -641.541,Z 463.297,A 0.000,B 0.000,C 90.000,E1 89.427} C_DIS
LIN {X 0.046,Y -640.692,Z 463.294,A 0.000,B 0.000,C 90.000,E1 88.912} C_DIS
LIN {X -0.192,Y -640.076,Z 463.293,A 0.000,B 0.000,C 90.000,E1 88.682} C_DIS
LIN {X 0.208,Y -639.288,Z 463.291,A 0.000,B 0.000,C 90.000,E1 88.396} C_DIS
LIN {X -0.256,Y -637.346,Z 463.288,A 0.000,B 0.000,C 90.000,E1 87.936} C_DIS
LIN {X 0.136,Y -636.332,Z 463.287,A 0.000,B 0.000,C 90.000,E1 87.650} C_DIS
LIN {X 0.265,Y -633.867,Z 463.284,A 0.000,B 0.000,C 90.000,E1 87.135} C_DIS
LIN {X 0.001,Y -628.224,Z 463.279,A 0.000,B 0.000,C 90.000,E1 86.274} C_DIS
LIN {X 0.252,Y -625.538,Z 463.277,A 0.000,B 0.000,C 90.000,E1 85.869} C_DIS
LIN {X 0.294,Y -621.747,Z 463.274,A 0.000,B 0.000,C 90.000,E1 85.355} C_DIS
LIN {X 0.203,Y -615.904,Z 463.271,A 0.000,B 0.000,C 90.000,E1 84.723} C_DIS
LIN {X -0.305,Y -609.425,Z 463.267,A 0.000,B 0.000,C 90.000,E1 84.147} C_DIS
LIN {X 0.234,Y -604.909,Z 463.265,A 0.000,B 0.000,C 90.000,E1 83.742} C_DIS
LIN {X -0.300,Y -603.678,Z 463.265,A 0.000,B 0.000,C 90.000,E1 83.685} C_DIS
LIN {X -0.117,Y -597.286,Z 463.262,A 0.000,B 0.000,C 90.000,E1 83.223} C_DIS
LIN {X 0.135,Y -593.719,Z 463.261,A 0.000,B 0.000,C 90.000,E1 82.996} C_DIS
LIN {X -0.241,Y -591.332,Z 463.260,A 0.000,B 0.000,C 90.000,E1 82.875} C_DIS
LIN {X -0.305,Y -586.124,Z 463.259,A 0.000,B 0.000,C 90.000,E1 82.591} C_DIS
LIN {X -0.159,Y -582.097,Z 463.258,A 0.000,B 0.000,C 90.000,E1 82.413} C_DIS
LIN {X 0.185,Y -577.625,Z 463.257,A 0.000,B 0.000,C 90.000,E1 82.186} C_DIS
LIN {X -0.010,Y -573.830,Z 463.256,A 0.000,B 0.000,C 90.000,E1 82.064} C_DIS
LIN {X -0.100,Y -567.254,Z 463.255,A 0.000,B 0.000,C 90.000,E1 81.894} C_DIS
LIN {X 0.256,Y -562.207,Z 463.255,A 0.000,B 0.000,C 90.000,E1 81.781} C_DIS
LIN {X -0.143,Y -557.503,Z 463.254,A 0.000,B 0.000,C 90.000,E1 81.781} C_DIS
LIN {X 0.241,Y -554.337,Z 463.254,A 0.000,B 0.000,C 90.000,E1 81.724} C_DIS
LIN {X 0.161,Y -484.693,Z 463.254,A 0.000,B 0.000,C 90.000,E1 81.724} C_DIS
LIN {X -0.070,Y -484.521,Z 463.252,A 0.000,B 0.000,C 90.000,E1 81.432} C_DIS
LIN {X -0.199,Y -480.458,Z 463.227,A 0.000,B 0.000,C 90.000,E1 76.825} C_DIS
LIN {X 0.150,Y -474.220,Z 463.201,A 0.000,B 0.000,C 90.000,E1 72.127} C_DIS
LIN {X 0.117,Y -473.712,Z 463.199,A 0.000,B 0.000,C 90.000,E1 71.819} C_DIS
LIN {X 0.239,Y -466.165,Z 463.175,A 0.000,B 0.000,C 90.000,E1 67.411} C_DIS
LIN {X 0.182,Y -465.738,Z 463.173,A 0.000,B 0.000,C 90.000,E1 67.102} C_DIS
LIN {X 0.049,Y -462.232,Z 463.164,A 0.000,B 0.000,C 90.000,E1 65.537} C_DIS
LIN {X -0.013,Y -457.839,Z 463.152,A 0.000,B 0.000,C 90.000,E1 63.307} C_DIS
LIN {X -0.053,Y -457.836,Z 463.152,A 0.000,B 0.000,C 90.000,E1 63.307} C_DIS
LIN {X 0.127,Y -466.130,Z 463.145,A 0.000,B 0.000,C 90.000,E1 62.025} C_DIS
LIN {X -0.053,Y -472.109,Z 463.139,A 0.000,B 0.000,C 90.000,E1 61.101} C_DIS
LIN {X 0.021,Y -478.765,Z 463.133,A 0.000,B 0.000,C 90.000,E1 59.999} C_DIS
LIN {X 0.203,Y -482.961,Z 463.129,A 0.000,B 0.000,C 90.000,E1 59.203} C_DIS
LIN {X 0.200,Y -485.322,Z 463.127,A 0.000,B 0.000,C 90.000,E1 58.742} C_DIS
LIN {X 0.028,Y -488.659,Z 463.122,A 0.000,B 0.000,C 90.000,E1 57.995} C_DIS
LIN {X 0.101,Y -491.043,Z 463.119,A 0.000,B 0.000,C 90.000,E1 57.375} C_DIS
LIN {X -0.079,Y -493.051,Z 463.115,A 0.000,B 0.000,C 90.000,E1 56.786} C_DIS
LIN {X -0.124,Y -495.525,Z 463.110,A 0.000,B 0.000,C 90.000,E1 55.881} C_DIS
LIN {X -0.002,Y -496.773,Z 463.107,A 0.000,B 0.000,C 90.000,E1 55.261} C_DIS
LIN {X -0.005,Y -498.183,Z 463.102,A 0.000,B 0.000,C 90.000,E1 54.356} C_DIS
LIN {X 0.301,Y -499.279,Z 463.097,A 0.000,B 0.000,C 90.000,E1 53.417} C_DIS
LIN {X -0.077,Y -499.939,Z 463.092,A 0.000,B 0.000,C 90.000,E1 52.557} C_DIS
LIN {X 0.253,Y -500.358,Z 463.087,A 0.000,B 0.000,C 90.000,E1 51.618} C_DIS
LIN {X 0.072,Y -500.538,Z 463.080,A 0.000,B 0.000,C 90.000,E1 50.436} C_DIS
LIN {X 0.144,Y -500.564,Z 463.077,A 0.000,B 0.000,C 90.000,E1 49.828} C_DIS
LIN {X -0.040,Y -500.243,Z 463.070,A 0.000,B 0.000,C 90.000,E1 48.647} C_DIS
LIN {X -0.274,Y -499.828,Z 463.064,A 0.000,B 0.000,C 90.000,E1 47.472} C_DIS
LIN {X -0.309,Y -499.132,Z 463.055,A 0.000,B 0.000,C 90.000,E1 45.972} C_DIS
LIN {X -0.208,Y -498.439,Z 463.049,A 0.000,B 0.000,C 90.000,E1 44.757} C_DIS
LIN {X 0.075,Y -497.431,Z 463.040,A 0.000,B 0.000,C 90.000,E1 43.218} C_DIS
LIN {X 0.167,Y -496.530,Z 463.033,A 0.000,B 0.000,C 90.000,E1 42.000} C_DIS
LIN {X -0.089,Y -495.068,Z 463.023,A 0.000,B 0.000,C 90.000,E1 40.216} C_DIS
LIN {X 0.053,Y -493.539,Z 463.013,A 0.000,B 0.000,C 90.000,E1 38.382} C_DIS
LIN {X 0.011,Y -492.225,Z 463.005,A 0.000,B 0.000,C 90.000,E1 36.870} C_DIS
LIN {X 0.094,Y -491.111,Z 462.998,A 0.000,B 0.000,C 90.000,E1 35.644} C_DIS
LIN {X -0.049,Y -489.177,Z 462.988,A 0.000,B 0.000,C 90.000,E1 33.833} C_DIS
LIN {X 0.078,Y -487.464,Z 462.979,A 0.000,B 0.000,C 90.000,E1 32.291} C_DIS
LIN {X -0.052,Y -485.986,Z 462.973,A 0.000,B 0.000,C 90.000,E1 31.082} C_DIS
LIN {X -0.206,Y -484.468,Z 462.966,A 0.000,B 0.000,C 90.000,E1 29.873} C_DIS
LIN {X -0.202,Y -481.826,Z 462.954,A 0.000,B 0.000,C 90.000,E1 27.719} C_DIS
LIN {X 0.115,Y -478.670,Z 462.938,A 0.000,B 0.000,C 90.000,E1 24.899} C_DIS
LIN {X -0.295,Y -475.999,Z 462.921,A 0.000,B 0.000,C 90.000,E1 21.844} C_DIS
LIN {X -0.017,Y -474.547,Z 462.909,A 0.000,B 0.000,C 90.000,E1 19.631} C_DIS
LIN {X -0.102,Y -473.225,Z 462.897,A 0.000,B 0.000,C 90.000,E1 17.457} C_DIS
LIN {X -0.092,Y -471.617,Z 462.883,A 0.000,B 0.000,C 90.000,E1 14.954} C_DIS
LIN {X 0.019,Y -470.169,Z 462.867,A 0.000,B 0.000,C 90.000,E1 12.119} C_DIS
LIN {X -0.237,Y -469.727,Z 462.860,A 0.000,B 0.000,C 90.000,E1 10.894} C_DIS
LIN {X -0.096,Y -469.151,Z 462.845,A 0.000,B 0.000,C 90.000,E1 8.049} C_DIS
LIN {X -0.071,Y -469.291,Z 462.826,A 0.000,B 0.000,C 90.000,E1 4.588} C_DIS
LIN {X -0.182,Y -470.702,Z 462.806,A 0.000,B 0.000,C 90.000,E1 1.146} C_DIS
LIN {X 0.020,Y -472.806,Z 462.790,A 0.000,B 0.000,C 90.000,E1 358.224} C_DIS
LIN {X -0.224,Y -475.315,Z 462.776,A 0.000,B 0.000,C 90.000,E1 355.755} C_DIS
LIN {X 0.133,Y -478.310,Z 462.762,A 0.000,B 0.000,C 90.000,E1 353.223} C_DIS
LIN {X -0.111,Y -481.284,Z 462.750,A 0.000,B 0.000,C 90.000,E1 351.084} C_DIS
LIN {X 0.013,Y -484.144,Z 462.740,A 0.000,B 0.000,C 90.000,E1 349.218} C_DIS
LIN {X 0.089,Y -491.591,Z 462.718,A 0.000,B 0.000,C 90.000,E1 345.227} C_DIS
LIN {X 0.163,Y -497.723,Z 462.703,A 0.000,B 0.000,C 90.000,E1 342.489} C_DIS
LIN {X -0.268,Y -502.114,Z 462.693,A 0.000,B 0.000,C 90.000,E1 340.732} C_DIS
LIN {X -0.131,Y -505.185,Z 462.686,A 0.000,B 0.000,C 90.000,E1 339.518} C_DIS
LIN {X -0.038,Y -509.716,Z 462.676,A 0.000,B 0.000,C 90.000,E1 337.720} C_DIS
LIN {X 0.162,Y -514.229,Z 462.666,A 0.000,B 0.000,C 90.000,E1 335.921} C_DIS
LIN {X 0.197,Y -518.629,Z 462.657,A 0.000,B 0.000,C 90.000,E1 334.152} C_DIS
LIN {X -0.288,Y -522.324,Z 462.648,A 0.000,B 0.000,C 90.000,E1 332.743} C_DIS
LIN {X 0.082,Y -527.423,Z 462.637,A 0.000,B 0.000,C 90.000,E1 330.667} C_DIS
LIN {X -0.072,Y -532.658,Z 462.626,A 0.000,B 0.000,C 90.000,E1 328.663} C_DIS
LIN {X 0.192,Y -537.164,Z 462.616,A 0.000,B 0.000,C 90.000,E1 326.914} C_DIS
LIN {X -0.066,Y -540.914,Z 462.608,A 0.000,B 0.000,C 90.000,E1 325.515} C_DIS
LIN {X -0.142,Y -547.066,Z 462.596,A 0.000,B 0.000,C 90.000,E1 323.256} C_DIS
LIN {X 0.160,Y -551.774,Z 462.586,A 0.000,B 0.000,C 90.000,E1 321.537} C_DIS
LIN {X -0.240,Y -557.151,Z 462.576,A 0.000,B 0.000,C 90.000,E1 319.622} C_DIS
LIN {X 0.130,Y -561.850,Z 462.566,A 0.000,B 0.000,C 90.000,E1 317.919} C_DIS
LIN {X -0.192,Y -566.462,Z 462.557,A 0.000,B 0.000,C 90.000,E1 316.296} C_DIS
LIN {X -0.137,Y -570.299,Z 462.550,A 0.000,B 0.000,C 90.000,E1 314.919} C_DIS
LIN {X 0.111,Y -574.809,Z 462.540,A 0.000,B 0.000,C 90.000,E1 313.257} C_DIS
LIN {X 0.067,Y -579.354,Z 462.531,A 0.000,B 0.000,C 90.000,E1 311.634} C_DIS
LIN {X 0.112,Y -583.753,Z 462.522,A 0.000,B 0.000,C 90.000,E1 310.011} C_DIS
LIN {X -0.071,Y -586.771,Z 462.516,A 0.000,B 0.000,C 90.000,E1 308.955} C_DIS
LIN {X -0.122,Y -589.635,Z 462.510,A 0.000,B 0.000,C 90.000,E1 307.890} C_DIS
LIN {X 0.094,Y -593.206,Z 462.503,A 0.000,B 0.000,C 90.000,E1 306.537} C_DIS
LIN {X -0.112,Y -596.719,Z 462.496,A 0.000,B 0.000,C 90.000,E1 305.231} C_DIS
LIN {X -0.127,Y -600.103,Z 462.488,A 0.000,B 0.000,C 90.000,E1 303.913} C_DIS
LIN {X -0.167,Y -603.869,Z 462.480,A 0.000,B 0.000,C 90.000,E1 302.339} C_DIS
LIN {X 0.067,Y -607.456,Z 462.471,A 0.000,B 0.000,C 90.000,E1 300.747} C_DIS
LIN {X -0.056,Y -609.673,Z 462.465,A 0.000,B 0.000,C 90.000,E1 299.716} C_DIS
LIN {X -0.229,Y -611.768,Z 462.459,A 0.000,B 0.000,C 90.000,E1 298.693} C_DIS
LIN {X -0.180,Y -615.833,Z 462.448,A 0.000,B 0.000,C 90.000,E1 296.616} C_DIS
LIN {X -0.257,Y -617.687,Z 462.442,A 0.000,B 0.000,C 90.000,E1 295.591} C_DIS
LIN {X 0.247,Y -619.367,Z 462.436,A 0.000,B 0.000,C 90.000,E1 294.515} C_DIS
LIN {X -0.055,Y -621.323,Z 462.429,A 0.000,B 0.000,C 90.000,E1 293.259} C_DIS
LIN {X 0.248,Y -622.759,Z 462.424,A 0.000,B 0.000,C 90.000,E1 292.206} C_DIS
LIN {X -0.236,Y -624.134,Z 462.418,A 0.000,B 0.000,C 90.000,E1 291.227} C_DIS
LIN {X 0.102,Y -625.405,Z 462.412,A 0.000,B 0.000,C 90.000,E1 290.174} C_DIS
LIN {X 0.238,Y -626.657,Z 462.407,A 0.000,B 0.000,C 90.000,E1 289.141} C_DIS
LIN {X -0.024,Y -628.305,Z 462.398,A 0.000,B 0.000,C 90.000,E1 287.638} C_DIS
LIN {X 0.350,Y -629.732,Z 462.390,A 0.000,B 0.000,C 90.000,E1 286.079} C_DIS
LIN {X 0.185,Y -630.513,Z 462.384,A 0.000,B 0.000,C 90.000,E1 285.079} C_DIS
LIN {X 0.009,Y -631.402,Z 462.377,A 0.000,B 0.000,C 90.000,E1 283.828} C_DIS
LIN {X -0.314,Y -632.027,Z 462.370,A 0.000,B 0.000,C 90.000,E1 282.591} C_DIS
LIN {X -0.015,Y -632.484,Z 462.363,A 0.000,B 0.000,C 90.000,E1 281.299} C_DIS
LIN {X -0.270,Y -632.682,Z 462.357,A 0.000,B 0.000,C 90.000,E1 280.310} C_DIS
LIN {X 0.245,Y -632.678,Z 462.349,A 0.000,B 0.000,C 90.000,E1 278.746} C_DIS
LIN {X -0.292,Y -632.321,Z 462.342,A 0.000,B 0.000,C 90.000,E1 277.530} C_DIS
LIN {X 0.068,Y -631.793,Z 462.336,A 0.000,B 0.000,C 90.000,E1 276.486} C_DIS
LIN {X 0.060,Y -630.807,Z 462.329,A 0.000,B 0.000,C 90.000,E1 275.220} C_DIS
LIN {X 0.266,Y -629.680,Z 462.323,A 0.000,B 0.000,C 90.000,E1 274.188} C_DIS
LIN {X -0.166,Y -628.329,Z 462.318,A 0.000,B 0.000,C 90.000,E1 273.212} C_DIS
LIN {X -0.266,Y -626.323,Z 462.311,A 0.000,B 0.000,C 90.000,E1 271.949} C_DIS
LIN {X 0.217,Y -624.025,Z 462.304,A 0.000,B 0.000,C 90.000,E1 270.630} C_DIS
LIN {X -0.309,Y -622.075,Z 462.298,A 0.000,B 0.000,C 90.000,E1 269.656} C_DIS
LIN {X -0.240,Y -620.054,Z 462.292,A 0.000,B 0.000,C 90.000,E1 268.625} C_DIS
LIN {X 0.120,Y -618.378,Z 462.288,A 0.000,B 0.000,C 90.000,E1 267.822} C_DIS
LIN {X -0.151,Y -615.498,Z 462.281,A 0.000,B 0.000,C 90.000,E1 266.560} C_DIS
LIN {X -0.153,Y -613.062,Z 462.275,A 0.000,B 0.000,C 90.000,E1 265.527} C_DIS
LIN {X -0.137,Y -610.552,Z 462.269,A 0.000,B 0.000,C 90.000,E1 264.489} C_DIS
LIN {X -0.170,Y -606.675,Z 462.261,A 0.000,B 0.000,C 90.000,E1 262.932} C_DIS
LIN {X 0.077,Y -603.366,Z 462.253,A 0.000,B 0.000,C 90.000,E1 261.602} C_DIS
LIN {X 0.268,Y -598.537,Z 462.243,A 0.000,B 0.000,C 90.000,E1 259.746} C_DIS
LIN {X -0.132,Y -594.871,Z 462.236,A 0.000,B 0.000,C 90.000,E1 258.465} C_DIS
LIN {X -0.203,Y -590.314,Z 462.227,A 0.000,B 0.000,C 90.000,E1 256.881} C_DIS
LIN {X -0.226,Y -585.657,Z 462.218,A 0.000,B 0.000,C 90.000,E1 255.283} C_DIS
LIN {X -0.013,Y -581.691,Z 462.211,A 0.000,B 0.000,C 90.000,E1 253.921} C_DIS
LIN {X 0.078,Y -578.499,Z 462.205,A 0.000,B 0.000,C 90.000,E1 252.834} C_DIS
LIN {X -0.041,Y -573.547,Z 462.196,A 0.000,B 0.000,C 90.000,E1 251.221} C_DIS
LIN {X 0.098,Y -568.370,Z 462.187,A 0.000,B 0.000,C 90.000,E1 249.571} C_DIS
LIN {X -0.202,Y -563.913,Z 462.179,A 0.000,B 0.000,C 90.000,E1 248.230} C_DIS
LIN {X 0.046,Y -560.160,Z 462.173,A 0.000,B 0.000,C 90.000,E1 247.102} C_DIS
LIN {X 0.019,Y -556.215,Z 462.167,A 0.000,B 0.000,C 90.000,E1 245.997} C_DIS
LIN {X -0.113,Y -552.205,Z 462.161,A 0.000,B 0.000,C 90.000,E1 244.897} C_DIS
LIN {X -0.019,Y -546.080,Z 462.151,A 0.000,B 0.000,C 90.000,E1 243.204} C_DIS
LIN {X -0.067,Y -538.930,Z 462.140,A 0.000,B 0.000,C 90.000,E1 241.229} C_DIS
LIN {X -0.256,Y -532.853,Z 462.131,A 0.000,B 0.000,C 90.000,E1 239.537} C_DIS
LIN {X -0.045,Y -526.775,Z 462.121,A 0.000,B 0.000,C 90.000,E1 237.788} C_DIS
LIN {X 0.312,Y -520.833,Z 462.111,A 0.000,B 0.000,C 90.000,E1 236.008} C_DIS
LIN {X -0.195,Y -516.788,Z 462.105,A 0.000,B 0.000,C 90.000,E1 234.895} C_DIS
LIN {X -0.193,Y -510.534,Z 462.095,A 0.000,B 0.000,C 90.000,E1 233.130} C_DIS
LIN {X -0.080,Y -499.111,Z 462.075,A 0.000,B 0.000,C 90.000,E1 229.542} C_DIS
LIN {X 0.072,Y -493.770,Z 462.065,A 0.000,B 0.000,C 90.000,E1 227.715} C_DIS
LIN {X 0.235,Y -487.784,Z 462.053,A 0.000,B 0.000,C 90.000,E1 225.567} C_DIS
LIN {X -0.103,Y -481.938,Z 462.041,A 0.000,B 0.000,C 90.000,E1 223.461} C_DIS
LIN {X -0.013,Y -477.140,Z 462.031,A 0.000,B 0.000,C 90.000,E1 221.595} C_DIS
LIN {X 0.098,Y -471.883,Z 462.019,A 0.000,B 0.000,C 90.000,E1 219.402} C_DIS
LIN {X 0.076,Y -467.545,Z 462.009,A 0.000,B 0.000,C 90.000,E1 217.523} C_DIS
LIN {X -0.044,Y -463.480,Z 461.998,A 0.000,B 0.000,C 90.000,E1 215.644} C_DIS
LIN {X -0.283,Y -460.827,Z 461.991,A 0.000,B 0.000,C 90.000,E1 214.405} C_DIS
LIN {X 0.036,Y -456.367,Z 461.979,A 0.000,B 0.000,C 90.000,E1 212.133} C_DIS
LIN {X 0.134,Y -452.063,Z 461.966,A 0.000,B 0.000,C 90.000,E1 209.873} C_DIS
LIN {X -0.181,Y -448.370,Z 461.955,A 0.000,B 0.000,C 90.000,E1 207.975} C_DIS
LIN {X -0.249,Y -445.296,Z 461.946,A 0.000,B 0.000,C 90.000,E1 206.360} C_DIS
LIN {X 0.118,Y -440.835,Z 461.934,A 0.000,B 0.000,C 90.000,E1 204.027} C_DIS
LIN {X 0.179,Y -436.345,Z 461.921,A 0.000,B 0.000,C 90.000,E1 201.716} C_DIS
LIN {X -0.030,Y -432.700,Z 461.910,A 0.000,B 0.000,C 90.000,E1 199.758} C_DIS
LIN {X 0.157,Y -428.702,Z 461.897,A 0.000,B 0.000,C 90.000,E1 197.402} C_DIS
LIN {X -0.048,Y -424.067,Z 461.880,A 0.000,B 0.000,C 90.000,E1 194.411} C_DIS
LIN {X 0.190,Y -421.259,Z 461.869,A 0.000,B 0.000,C 90.000,E1 192.355} C_DIS
LIN {X -0.012,Y -417.872,Z 461.854,A 0.000,B 0.000,C 90.000,E1 189.670} C_DIS
LIN {X -0.095,Y -415.096,Z 461.841,A 0.000,B 0.000,C 90.000,E1 187.296} C_DIS
LIN {X 0.029,Y -413.285,Z 461.831,A 0.000,B 0.000,C 90.000,E1 185.568} C_DIS
LIN {X 0.117,Y -410.338,Z 461.814,A 0.000,B 0.000,C 90.000,E1 182.465} C_DIS
LIN {X 0.059,Y -408.288,Z 461.798,A 0.000,B 0.000,C 90.000,E1 179.714} C_DIS
LIN {X -0.062,Y -406.869,Z 461.783,A 0.000,B 0.000,C 90.000,E1 176.963} C_DIS
LIN {X -0.191,Y -405.945,Z 461.764,A 0.000,B 0.000,C 90.000,E1 173.514} C_DIS
LIN {X -0.150,Y -406.169,Z 461.745,A 0.000,B 0.000,C 90.000,E1 170.038} C_DIS
LIN {X -0.169,Y -407.490,Z 461.723,A 0.000,B 0.000,C 90.000,E1 166.228} C_DIS
LIN {X 0.074,Y -408.400,Z 461.714,A 0.000,B 0.000,C 90.000,E1 164.464} C_DIS
LIN {X 0.004,Y -411.214,Z 461.693,A 0.000,B 0.000,C 90.000,E1 160.678} C_DIS
LIN {X -0.037,Y -414.274,Z 461.676,A 0.000,B 0.000,C 90.000,E1 157.592} C_DIS
LIN {X 0.056,Y -417.474,Z 461.660,A 0.000,B 0.000,C 90.000,E1 154.845} C_DIS
LIN {X 0.170,Y -419.597,Z 461.651,A 0.000,B 0.000,C 90.000,E1 153.127} C_DIS
LIN {X -0.125,Y -422.767,Z 461.638,A 0.000,B 0.000,C 90.000,E1 150.795} C_DIS
LIN {X 0.076,Y -425.946,Z 461.625,A 0.000,B 0.000,C 90.000,E1 148.408} C_DIS
LIN {X -0.135,Y -429.329,Z 461.612,A 0.000,B 0.000,C 90.000,E1 146.087} C_DIS
LIN {X -0.019,Y -432.372,Z 461.600,A 0.000,B 0.000,C 90.000,E1 144.069} C_DIS
LIN {X 0.069,Y -434.958,Z 461.591,A 0.000,B 0.000,C 90.000,E1 142.396} C_DIS
LIN {X 0.161,Y -438.720,Z 461.578,A 0.000,B 0.000,C 90.000,E1 140.070} C_DIS
LIN {X -0.013,Y -442.016,Z 461.567,A 0.000,B 0.000,C 90.000,E1 138.119} C_DIS
LIN {X -0.128,Y -444.089,Z 461.560,A 0.000,B 0.000,C 90.000,E1 136.824} C_DIS
LIN {X 0.122,Y -445.977,Z 461.553,A 0.000,B 0.000,C 90.000,E1 135.486} C_DIS
LIN {X 0.080,Y -447.473,Z 461.546,A 0.000,B 0.000,C 90.000,E1 134.190} C_DIS
LIN {X 0.054,Y -448.640,Z 461.538,A 0.000,B 0.000,C 90.000,E1 132.894} C_DIS
LIN {X 0.069,Y -449.253,Z 461.533,A 0.000,B 0.000,C 90.000,E1 131.919} C_DIS
LIN {X 0.099,Y -449.597,Z 461.528,A 0.000,B 0.000,C 90.000,E1 130.943} C_DIS
LIN {X 0.089,Y -449.572,Z 461.524,A 0.000,B 0.000,C 90.000,E1 130.297} C_DIS
LIN {X 0.130,Y -449.426,Z 461.520,A 0.000,B 0.000,C 90.000,E1 129.644} C_DIS
LIN {X 0.158,Y -448.811,Z 461.515,A 0.000,B 0.000,C 90.000,E1 128.669} C_DIS
LIN {X -0.100,Y -447.845,Z 461.510,A 0.000,B 0.000,C 90.000,E1 127.729} C_DIS
LIN {X -0.011,Y -446.620,Z 461.504,A 0.000,B 0.000,C 90.000,E1 126.744} C_DIS
LIN {X 0.069,Y -445.166,Z 461.499,A 0.000,B 0.000,C 90.000,E1 125.758} C_DIS
LIN {X 0.072,Y -442.631,Z 461.492,A 0.000,B 0.000,C 90.000,E1 124.452} C_DIS
LIN {X -0.150,Y -440.440,Z 461.486,A 0.000,B 0.000,C 90.000,E1 123.499} C_DIS
LIN {X 0.281,Y -436.460,Z 461.477,A 0.000,B 0.000,C 90.000,E1 121.799} C_DIS
LIN {X 0.009,Y -433.118,Z 461.470,A 0.000,B 0.000,C 90.000,E1 120.512} C_DIS
LIN {X 0.074,Y -431.589,Z 461.466,A 0.000,B 0.000,C 90.000,E1 119.922} C_DIS
LIN {X 0.035,Y -431.579,Z 461.466,A 0.000,B 0.000,C 90.000,E1 119.922} C_DIS
LIN {X -0.198,Y -441.014,Z 461.446,A 0.000,B 0.000,C 90.000,E1 116.232} C_DIS
LIN {X -0.034,Y -444.867,Z 461.438,A 0.000,B 0.000,C 90.000,E1 114.899} C_DIS
LIN {X 0.225,Y -453.976,Z 461.417,A 0.000,B 0.000,C 90.000,E1 110.972} C_DIS
LIN {X 0.083,Y -457.444,Z 461.410,A 0.000,B 0.000,C 90.000,E1 109.704} C_DIS
LIN {X 0.185,Y -466.099,Z 461.387,A 0.000,B 0.000,C 90.000,E1 105.552} C_DIS
LIN {X -0.091,Y -467.669,Z 461.383,A 0.000,B 0.000,C 90.000,E1 104.954} C_DIS
LIN {X -0.134,Y -475.884,Z 461.357,A 0.000,B 0.000,C 90.000,E1 100.254} C_DIS
LIN {X 0.173,Y -476.342,Z 461.355,A 0.000,B 0.000,C 90.000,E1 99.905} C_DIS
LIN {X -0.069,Y -478.665,Z 461.343,A 0.000,B 0.000,C 90.000,E1 97.814} C_DIS
LIN {X -0.128,Y -553.443,Z 461.343,A 0.000,B 0.000,C 90.000,E1 97.814} C_DIS
LIN {X 0.231,Y -560.012,Z 461.343,A 0.000,B 0.000,C 90.000,E1 97.701} C_DIS
LIN {X -0.096,Y -565.501,Z 461.342,A 0.000,B 0.000,C 90.000,E1 97.644} C_DIS
LIN {X 0.226,Y -571.711,Z 461.342,A 0.000,B 0.000,C 90.000,E1 97.473} C_DIS
LIN {X 0.226,Y -578.097,Z 461.341,A 0.000,B 0.000,C 90.000,E1 97.296} C_DIS
LIN {X -0.227,Y -584.603,Z 461.340,A 0.000,B 0.000,C 90.000,E1 97.125} C_DIS
LIN {X 0.248,Y -590.977,Z 461.338,A 0.000,B 0.000,C 90.000,E1 96.834} C_DIS
LIN {X 0.258,Y -597.043,Z 461.337,A 0.000,B 0.000,C 90.000,E1 96.549} C_DIS
LIN {X -0.064,Y -603.100,Z 461.335,A 0.000,B 0.000,C 90.000,E1 96.258} C_DIS
LIN {X -0.212,Y -608.904,Z 461.333,A 0.000,B 0.000,C 90.000,E1 95.910} C_DIS
LIN {X -0.264,Y -614.510,Z 461.331,A 0.000,B 0.000,C 90.000,E1 95.511} C_DIS
LIN {X -0.119,Y -620.813,Z 461.327,A 0.000,B 0.000,C 90.000,E1 94.935} C_DIS
LIN {X -0.241,Y -623.071,Z 461.326,A 0.000,B 0.000,C 90.000,E1 94.702} C_DIS
LIN {X -0.186,Y -627.544,Z 461.323,A 0.000,B 0.000,C 90.000,E1 94.188} C_DIS
LIN {X -0.222,Y -631.437,Z 461.320,A 0.000,B 0.000,C 90.000,E1 93.555} C_DIS
LIN {X -0.096,Y -634.289,Z 461.317,A 0.000,B 0.000,C 90.000,E1 93.037} C_DIS
LIN {X 0.015,Y -636.048,Z 461.314,A 0.000,B 0.000,C 90.000,E1 92.522} C_DIS
LIN {X -0.088,Y -638.311,Z 461.310,A 0.000,B 0.000,C 90.000,E1 91.776} C_DIS
LIN {X 0.053,Y -639.356,Z 461.307,A 0.000,B 0.000,C 90.000,E1 91.260} C_DIS
LIN {X 0.205,Y -639.902,Z 461.304,A 0.000,B 0.000,C 90.000,E1 90.745} C_DIS
LIN {X -0.037,Y -640.015,Z 461.303,A 0.000,B 0.000,C 90.000,E1 90.516} C_DIS
LIN {X 0.123,Y -639.950,Z 461.300,A 0.000,B 0.000,C 90.000,E1 90.000} C_DIS
LIN {X 0.282,Y -639.363,Z 461.297,A 0.000,B 0.000,C 90.000,E1 89.484} C_DIS
LIN {X -0.201,Y -638.198,Z 461.295,A 0.000,B 0.000,C 90.000,E1 89.026} C_DIS
LIN {X -0.055,Y -636.696,Z 461.292,A 0.000,B 0.000,C 90.000,E1 88.511} C_DIS
LIN {X -0.304,Y -635.873,Z 461.290,A 0.000,B 0.000,C 90.000,E1 88.282} C_DIS
LIN {X -0.278,Y -633.333,Z 461.287,A 0.000,B 0.000,C 90.000,E1 87.650} C_DIS
LIN {X 0.087,Y -627.849,Z 461.282,A 0.000,B 0.000,C 90.000,E1 86.731} C_DIS
LIN {X 0.294,Y -625.218,Z 461.280,A 0.000,B 0.000,C 90.000,E1 86.331} C_DIS
LIN {X -0.239,Y -621.521,Z 461.277,A 0.000,B 0.000,C 90.000,E1 85.869} C_DIS
LIN {X 0.239,Y -615.945,Z 461.273,A 0.000,B 0.000,C 90.000,E1 85.184} C_DIS
LIN {X -0.171,Y -610.755,Z 461.271,A 0.000,B 0.000,C 90.000,E1 84.723} C_DIS
LIN {X -0.281,Y -608.026,Z 461.269,A 0.000,B 0.000,C 90.000,E1 84.489} C_DIS
LIN {X -0.308,Y -603.772,Z 461.267,A 0.000,B 0.000,C 90.000,E1 84.147} C_DIS
LIN {X -0.174,Y -600.607,Z 461.266,A 0.000,B 0.000,C 90.000,E1 83.913} C_DIS
LIN {X 0.180,Y -595.873,Z 461.264,A 0.000,B 0.000,C 90.000,E1 83.571} C_DIS
LIN {X 0.230,Y -591.097,Z 461.263,A 0.000,B 0.000,C 90.000,E1 83.280} C_DIS
LIN {X 0.250,Y -584.248,Z 461.261,A 0.000,B 0.000,C 90.000,E1 82.932} C_DIS
LIN {X -0.224,Y -578.586,Z 461.260,A 0.000,B 0.000,C 90.000,E1 82.761} C_DIS
LIN {X 0.179,Y -572.920,Z 461.259,A 0.000,B 0.000,C 90.000,E1 82.534} C_DIS
LIN {X -0.222,Y -565.700,Z 461.258,A 0.000,B 0.000,C 90.000,E1 82.413} C_DIS
LIN {X -0.230,Y -559.434,Z 461.257,A 0.000,B 0.000,C 90.000,E1 82.356} C_DIS
LIN {X -0.232,Y -484.743,Z 461.257,A 0.000,B 0.000,C 90.000,E1 82.356} C_DIS
LIN {X -0.174,Y -484.676,Z 461.253,A 0.000,B 0.000,C 90.000,E1 81.602} C_DIS
LIN {X 0.194,Y -480.595,Z 461.228,A 0.000,B 0.000,C 90.000,E1 76.937} C_DIS
LIN {X -0.093,Y -479.694,Z 461.224,A 0.000,B 0.000,C 90.000,E1 76.353} C_DIS
LIN {X -0.059,Y -474.036,Z 461.200,A 0.000,B 0.000,C 90.000,E1 72.000} C_DIS
LIN {X -0.029,Y -465.460,Z 461.172,A 0.000,B 0.000,C 90.000,E1 66.975} C_DIS
LIN {X 0.136,Y -458.243,Z 461.153,A 0.000,B 0.000,C 90.000,E1 63.512} C_DIS
LIN {X 0.096,Y -458.250,Z 461.153,A 0.000,B 0.000,C 90.000,E1 63.512} C_DIS
LIN {X 0.043,Y -465.959,Z 461.147,A 0.000,B 0.000,C 90.000,E1 62.359} C_DIS
LIN {X -0.119,Y -472.153,Z 461.141,A 0.000,B 0.000,C 90.000,E1 61.435} C_DIS
LIN {X -0.025,Y -478.876,Z 461.135,A 0.000,B 0.000,C 90.000,E1 60.333} C_DIS
LIN {X 0.159,Y -483.283,Z 461.131,A 0.000,B 0.000,C 90.000,E1 59.537} C_DIS
LIN {X -0.064,Y -486.449,Z 461.128,A 0.000,B 0.000,C 90.000,E1 58.948} C_DIS
LIN {X -0.229,Y -489.873,Z 461.123,A 0.000,B 0.000,C 90.000,E1 58.201} C_DIS
LIN {X -0.148,Y -492.303,Z 461.120,A 0.000,B 0.000,C 90.000,E1 57.582} C_DIS
LIN {X -0.047,Y -494.343,Z 461.116,A 0.000,B 0.000,C 90.000,E1 56.962} C_DIS
LIN {X 0.069,Y -496.071,Z 461.113,A 0.000,B 0.000,C 90.000,E1 56.342} C_DIS
LIN {X 0.339,Y -496.890,Z 461.111,A 0.000,B 0.000,C 90.000,E1 56.008} C_DIS
LIN {X -0.217,Y -498.156,Z 461.108,A 0.000,B 0.000,C 90.000,E1 55.468} C_DIS
LIN {X -0.074,Y -499.135,Z 461.105,A 0.000,B 0.000,C 90.000,E1 54.848} C_DIS
LIN {X 0.118,Y -500.743,Z 461.098,A 0.000,B 0.000,C 90.000,E1 53.623} C_DIS
LIN {X -0.243,Y -501.400,Z 461.093,A 0.000,B 0.000,C 90.000,E1 52.763} C_DIS
LIN {X 0.107,Y -501.801,Z 461.088,A 0.000,B 0.000,C 90.000,E1 51.823} C_DIS
LIN {X -0.050,Y -501.964,Z 461.081,A 0.000,B 0.000,C 90.000,E1 50.642} C_DIS
LIN {X 0.033,Y -501.988,Z 461.078,A 0.000,B 0.000,C 90.000,E1 50.033} C_DIS
LIN {X -0.123,Y -501.605,Z 461.071,A 0.000,B 0.000,C 90.000,E1 48.852} C_DIS
LIN {X 0.244,Y -501.032,Z 461.063,A 0.000,B 0.000,C 90.000,E1 47.310} C_DIS
LIN {X 0.231,Y -500.211,Z 461.055,A 0.000,B 0.000,C 90.000,E1 45.810} C_DIS
LIN {X -0.007,Y -499.471,Z 461.048,A 0.000,B 0.000,C 90.000,E1 44.636} C_DIS
LIN {X -0.198,Y -498.161,Z 461.038,A 0.000,B 0.000,C 90.000,E1 42.852} C_DIS
LIN {X 0.102,Y -496.951,Z 461.030,A 0.000,B 0.000,C 90.000,E1 41.310} C_DIS
LIN {X 0.052,Y -495.699,Z 461.021,A 0.000,B 0.000,C 90.000,E1 39.806} C_DIS
LIN {X -0.169,Y -494.135,Z 461.011,A 0.000,B 0.000,C 90.000,E1 38.016} C_DIS
LIN {X -0.202,Y -492.793,Z 461.003,A 0.000,B 0.000,C 90.000,E1 36.503} C_DIS
LIN {X -0.248,Y -491.890,Z 460.998,A 0.000,B 0.000,C 90.000,E1 35.598} C_DIS
LIN {X 0.316,Y -489.929,Z 460.988,A 0.000,B 0.000,C 90.000,E1 33.706} C_DIS
LIN {X 0.047,Y -488.227,Z 460.979,A 0.000,B 0.000,C 90.000,E1 32.212} C_DIS
LIN {X -0.022,Y -485.974,Z 460.969,A 0.000,B 0.000,C 90.000,E1 30.384} C_DIS
LIN {X -0.210,Y -483.628,Z 460.959,A 0.000,B 0.000,C 90.000,E1 28.565} C_DIS
LIN {X -0.206,Y -482.501,Z 460.953,A 0.000,B 0.000,C 90.000,E1 27.641} C_DIS
LIN {X 0.123,Y -479.372,Z 460.938,A 0.000,B 0.000,C 90.000,E1 24.823} C_DIS
LIN {X 0.150,Y -476.464,Z 460.919,A 0.000,B 0.000,C 90.000,E1 21.408} C_DIS
LIN {X -0.147,Y -475.257,Z 460.909,A 0.000,B 0.000,C 90.000,E1 19.577} C_DIS
LIN {X -0.208,Y -473.919,Z 460.897,A 0.000,B 0.000,C 90.000,E1 17.402} C_DIS
LIN {X -0.171,Y -472.284,Z 460.883,A 0.000,B 0.000,C 90.000,E1 14.898} C_DIS
LIN {X -0.099,Y -470.503,Z 460.862,A 0.000,B 0.000,C 90.000,E1 11.130} C_DIS
LIN {X -0.108,Y -469.764,Z 460.844,A 0.000,B 0.000,C 90.000,E1 7.992} C_DIS
LIN {X -0.056,Y -469.889,Z 460.825,A 0.000,B 0.000,C 90.000,E1 4.531} C_DIS
LIN {X 0.108,Y -471.465,Z 460.804,A 0.000,B 0.000,C 90.000,E1 0.745} C_DIS
LIN {X 0.213,Y -472.565,Z 460.795,A 0.000,B 0.000,C 90.000,E1 359.141} C_DIS
LIN {X 0.199,Y -475.154,Z 460.780,A 0.000,B 0.000,C 90.000,E1 356.331} C_DIS
LIN {X -0.139,Y -478.450,Z 460.764,A 0.000,B 0.000,C 90.000,E1 353.571} C_DIS
LIN {X 0.091,Y -481.362,Z 460.752,A 0.000,B 0.000,C 90.000,E1 351.376} C_DIS
LIN {X 0.083,Y -484.696,Z 460.740,A 0.000,B 0.000,C 90.000,E1 349.218} C_DIS
LIN {X 0.188,Y -492.124,Z 460.718,A 0.000,B 0.000,C 90.000,E1 345.227} C_DIS
LIN {X -0.195,Y -498.305,Z 460.703,A 0.000,B 0.000,C 90.000,E1 342.543} C_DIS
LIN {X -0.062,Y -503.487,Z 460.691,A 0.000,B 0.000,C 90.000,E1 340.423} C_DIS
LIN {X 0.191,Y -507.307,Z 460.683,A 0.000,B 0.000,C 90.000,E1 338.901} C_DIS
LIN {X 0.120,Y -510.380,Z 460.676,A 0.000,B 0.000,C 90.000,E1 337.720} C_DIS
LIN {X -0.134,Y -514.918,Z 460.666,A 0.000,B 0.000,C 90.000,E1 335.973} C_DIS
LIN {X 0.254,Y -518.616,Z 460.658,A 0.000,B 0.000,C 90.000,E1 334.460} C_DIS
LIN {X -0.083,Y -523.119,Z 460.649,A 0.000,B 0.000,C 90.000,E1 332.743} C_DIS
LIN {X 0.002,Y -528.991,Z 460.636,A 0.000,B 0.000,C 90.000,E1 330.411} C_DIS
LIN {X -0.117,Y -534.279,Z 460.624,A 0.000,B 0.000,C 90.000,E1 328.408} C_DIS
LIN {X -0.275,Y -538.841,Z 460.615,A 0.000,B 0.000,C 90.000,E1 326.707} C_DIS
LIN {X -0.060,Y -542.605,Z 460.607,A 0.000,B 0.000,C 90.000,E1 325.261} C_DIS
LIN {X -0.147,Y -548.046,Z 460.596,A 0.000,B 0.000,C 90.000,E1 323.290} C_DIS
LIN {X -0.270,Y -552.778,Z 460.587,A 0.000,B 0.000,C 90.000,E1 321.618} C_DIS
LIN {X -0.211,Y -559.027,Z 460.574,A 0.000,B 0.000,C 90.000,E1 319.380} C_DIS
LIN {X -0.173,Y -563.788,Z 460.565,A 0.000,B 0.000,C 90.000,E1 317.715} C_DIS
LIN {X 0.240,Y -567.662,Z 460.557,A 0.000,B 0.000,C 90.000,E1 316.296} C_DIS
LIN {X 0.020,Y -572.284,Z 460.548,A 0.000,B 0.000,C 90.000,E1 314.676} C_DIS
LIN {X -0.110,Y -576.867,Z 460.539,A 0.000,B 0.000,C 90.000,E1 313.056} C_DIS
LIN {X 0.152,Y -580.720,Z 460.532,A 0.000,B 0.000,C 90.000,E1 311.676} C_DIS
LIN {X -0.162,Y -585.222,Z 460.523,A 0.000,B 0.000,C 90.000,E1 310.092} C_DIS
LIN {X -0.129,Y -588.997,Z 460.515,A 0.000,B 0.000,C 90.000,E1 308.749} C_DIS
LIN {X -0.191,Y -593.328,Z 460.506,A 0.000,B 0.000,C 90.000,E1 307.156} C_DIS
LIN {X 0.085,Y -596.871,Z 460.499,A 0.000,B 0.000,C 90.000,E1 305.804} C_DIS
LIN {X 0.078,Y -600.346,Z 460.492,A 0.000,B 0.000,C 90.000,E1 304.485} C_DIS
LIN {X 0.134,Y -603.599,Z 460.484,A 0.000,B 0.000,C 90.000,E1 303.166} C_DIS
LIN {X -0.023,Y -606.074,Z 460.479,A 0.000,B 0.000,C 90.000,E1 302.133} C_DIS
LIN {X 0.308,Y -609.076,Z 460.471,A 0.000,B 0.000,C 90.000,E1 300.797} C_DIS
LIN {X -0.100,Y -611.319,Z 460.466,A 0.000,B 0.000,C 90.000,E1 299.795} C_DIS
LIN {X 0.048,Y -613.440,Z 460.460,A 0.000,B 0.000,C 90.000,E1 298.743} C_DIS
LIN {X -0.040,Y -614.964,Z 460.455,A 0.000,B 0.000,C 90.000,E1 297.975} C_DIS
LIN {X -0.087,Y -615.964,Z 460.453,A 0.000,B 0.000,C 90.000,E1 297.462} C_DIS
LIN {X 0.103,Y -618.595,Z 460.445,A 0.000,B 0.000,C 90.000,E1 296.155} C_DIS
LIN {X -0.208,Y -620.388,Z 460.440,A 0.000,B 0.000,C 90.000,E1 295.155} C_DIS
LIN {X 0.336,Y -622.059,Z 460.434,A 0.000,B 0.000,C 90.000,E1 294.079} C_DIS
LIN {X 0.080,Y -624.015,Z 460.427,A 0.000,B 0.000,C 90.000,E1 292.823} C_DIS
LIN {X 0.191,Y -626.109,Z 460.418,A 0.000,B 0.000,C 90.000,E1 291.280} C_DIS
LIN {X -0.251,Y -627.432,Z 460.413,A 0.000,B 0.000,C 90.000,E1 290.301} C_DIS
LIN {X -0.292,Y -628.987,Z 460.406,A 0.000,B 0.000,C 90.000,E1 289.033} C_DIS
LIN {X -0.301,Y -630.398,Z 460.399,A 0.000,B 0.000,C 90.000,E1 287.764} C_DIS
LIN {X 0.121,Y -631.846,Z 460.390,A 0.000,B 0.000,C 90.000,E1 286.205} C_DIS
LIN {X 0.154,Y -632.665,Z 460.385,A 0.000,B 0.000,C 90.000,E1 285.190} C_DIS
LIN {X -0.176,Y -633.708,Z 460.376,A 0.000,B 0.000,C 90.000,E1 283.703} C_DIS
LIN {X 0.332,Y -634.200,Z 460.370,A 0.000,B 0.000,C 90.000,E1 282.647} C_DIS
LIN {X -0.083,Y -634.672,Z 460.363,A 0.000,B 0.000,C 90.000,E1 281.422} C_DIS
LIN {X -0.187,Y -634.885,Z 460.358,A 0.000,B 0.000,C 90.000,E1 280.423} C_DIS
LIN {X -0.074,Y -634.880,Z 460.351,A 0.000,B 0.000,C 90.000,E1 279.151} C_DIS
LIN {X -0.296,Y -634.735,Z 460.345,A 0.000,B 0.000,C 90.000,E1 278.163} C_DIS
LIN {X 0.020,Y -634.347,Z 460.340,A 0.000,B 0.000,C 90.000,E1 277.125} C_DIS
LIN {X -0.024,Y -633.909,Z 460.335,A 0.000,B 0.000,C 90.000,E1 276.372} C_DIS
LIN {X 0.277,Y -633.124,Z 460.330,A 0.000,B 0.000,C 90.000,E1 275.334} C_DIS
LIN {X 0.151,Y -632.308,Z 460.326,A 0.000,B 0.000,C 90.000,E1 274.588} C_DIS
LIN {X -0.252,Y -630.986,Z 460.320,A 0.000,B 0.000,C 90.000,E1 273.612} C_DIS
LIN {X 0.230,Y -629.859,Z 460.316,A 0.000,B 0.000,C 90.000,E1 272.808} C_DIS
LIN {X 0.044,Y -628.673,Z 460.312,A 0.000,B 0.000,C 90.000,E1 272.064} C_DIS
LIN {X -0.061,Y -626.313,Z 460.304,A 0.000,B 0.000,C 90.000,E1 270.802} C_DIS
LIN {X 0.067,Y -624.373,Z 460.299,A 0.000,B 0.000,C 90.000,E1 269.771} C_DIS
LIN {X -0.125,Y -621.743,Z 460.292,A 0.000,B 0.000,C 90.000,E1 268.511} C_DIS
LIN {X -0.046,Y -619.446,Z 460.286,A 0.000,B 0.000,C 90.000,E1 267.478} C_DIS
LIN {X 0.007,Y -617.086,Z 460.280,A 0.000,B 0.000,C 90.000,E1 266.445} C_DIS
LIN {X -0.245,Y -613.999,Z 460.273,A 0.000,B 0.000,C 90.000,E1 265.179} C_DIS
LIN {X -0.273,Y -611.409,Z 460.267,A 0.000,B 0.000,C 90.000,E1 264.147} C_DIS
LIN {X 0.051,Y -608.155,Z 460.260,A 0.000,B 0.000,C 90.000,E1 262.818} C_DIS
LIN {X -0.280,Y -604.753,Z 460.253,A 0.000,B 0.000,C 90.000,E1 261.546} C_DIS
LIN {X 0.229,Y -600.595,Z 460.244,A 0.000,B 0.000,C 90.000,E1 259.926} C_DIS
LIN {X 0.263,Y -597.640,Z 460.238,A 0.000,B 0.000,C 90.000,E1 258.870} C_DIS
LIN {X 0.124,Y -593.139,Z 460.230,A 0.000,B 0.000,C 90.000,E1 257.297} C_DIS
LIN {X -0.110,Y -589.219,Z 460.222,A 0.000,B 0.000,C 90.000,E1 255.992} C_DIS
LIN {X 0.168,Y -585.290,Z 460.215,A 0.000,B 0.000,C 90.000,E1 254.629} C_DIS
LIN {X 0.198,Y -580.427,Z 460.206,A 0.000,B 0.000,C 90.000,E1 253.015} C_DIS
LIN {X 0.119,Y -575.414,Z 460.197,A 0.000,B 0.000,C 90.000,E1 251.402} C_DIS
LIN {X 0.119,Y -571.970,Z 460.191,A 0.000,B 0.000,C 90.000,E1 250.315} C_DIS
LIN {X 0.081,Y -567.561,Z 460.183,A 0.000,B 0.000,C 90.000,E1 248.954} C_DIS
LIN {X 0.171,Y -563.908,Z 460.177,A 0.000,B 0.000,C 90.000,E1 247.847} C_DIS
LIN {X -0.113,Y -561.041,Z 460.172,A 0.000,B 0.000,C 90.000,E1 247.050} C_DIS
LIN {X 0.097,Y -557.064,Z 460.166,A 0.000,B 0.000,C 90.000,E1 245.921} C_DIS
LIN {X -0.254,Y -553.037,Z 460.160,A 0.000,B 0.000,C 90.000,E1 244.845} C_DIS
LIN {X -0.154,Y -547.905,Z 460.152,A 0.000,B 0.000,C 90.000,E1 243.435} C_DIS
LIN {X -0.184,Y -539.647,Z 460.140,A 0.000,B 0.000,C 90.000,E1 241.179} C_DIS
LIN {X -0.093,Y -533.544,Z 460.130,A 0.000,B 0.000,C 90.000,E1 239.459} C_DIS
LIN {X 0.136,Y -527.454,Z 460.121,A 0.000,B 0.000,C 90.000,E1 237.709} C_DIS
LIN {X -0.214,Y -521.453,Z 460.111,A 0.000,B 0.000,C 90.000,E1 236.008} C_DIS
LIN {X 0.013,Y -517.393,Z 460.105,A 0.000,B 0.000,C 90.000,E1 234.815} C_DIS
LIN {X 0.028,Y -511.152,Z 460.095,A 0.000,B 0.000,C 90.000,E1 233.050} C_DIS
LIN {X 0.169,Y -499.754,Z 460.075,A 0.000,B 0.000,C 90.000,E1 229.461} C_DIS
LIN {X -0.181,Y -493.552,Z 460.063,A 0.000,B 0.000,C 90.000,E1 227.391} C_DIS
LIN {X -0.178,Y -488.408,Z 460.053,A 0.000,B 0.000,C 90.000,E1 225.567} C_DIS
LIN {X 0.186,Y -482.583,Z 460.041,A 0.000,B 0.000,C 90.000,E1 223.380} C_DIS
LIN {X -0.030,Y -477.768,Z 460.031,A 0.000,B 0.000,C 90.000,E1 221.553} C_DIS
LIN {X -0.105,Y -471.784,Z 460.017,A 0.000,B 0.000,C 90.000,E1 219.072} C_DIS
LIN {X 0.117,Y -465.425,Z 460.001,A 0.000,B 0.000,C 90.000,E1 216.217} C_DIS
